SPLINE
SPL {X  -165.650, Y  +484.445, Z    +0.000, E1   +32.277, E3 +467467.662}
SPL {X  -165.650, Y  +481.524, Z    +0.000, E1   +31.089, E3 +467485.112}
SPL {X  -165.650, Y  +478.014, Z    +0.000, E1   +30.826, E3 +467498.720}
SPL {X  -165.650, Y  +474.473, Z    +0.000, E1   +30.943, E3 +467510.044}
SPL {X  -165.650, Y  +471.826, Z    +0.000, E1   +30.770, E3 +467520.228}
SPL {X  -165.650, Y  +467.753, Z    +0.000, E1   +30.878, E3 +467533.601}
SPL {X  -165.650, Y  +463.837, Z    +0.000, E1   +30.924, E3 +467546.535}
SPL {X  -165.650, Y  +461.106, Z    +0.000, E1   +30.916, E3 +467555.922}
SPL {X  -165.650, Y  +457.156, Z    +0.000, E1   +30.860, E3 +467569.999}
SPL {X  -165.650, Y  +453.156, Z    +0.000, E1   +30.934, E3 +467582.973}
SPL {X  -165.650, Y  +450.433, Z    +0.000, E1   +30.789, E3 +467593.328}
SPL {X  -165.650, Y  +447.097, Z    +0.000, E1   +30.843, E3 +467604.377}
SPL {X  -165.650, Y  +443.673, Z    +0.000, E1   +30.907, E3 +467615.684}
SPL {X  -165.650, Y  +439.486, Z    +0.000, E1   +30.857, E3 +467630.493}
SPL {X  -165.650, Y  +434.043, Z    +0.000, E1   +30.950, E3 +467648.510}
SPL {X  -165.650, Y  +430.419, Z    +0.000, E1   +30.895, E3 +467661.013}
SPL {X  -165.650, Y  +427.340, Z    +0.000, E1   +30.870, E3 +467671.839}
SPL {X  -165.650, Y  +422.641, Z    +0.000, E1   +30.884, E3 +467687.928}
SPL {X  -165.650, Y  +417.366, Z    +0.000, E1   +30.879, E3 +467706.034}
SPL {X  -165.650, Y  +412.139, Z    +0.000, E1   +30.870, E3 +467723.984}
SPL {X  -165.650, Y  +406.834, Z    +0.000, E1   +30.919, E3 +467741.812}
SPL {X  -165.650, Y  +402.516, Z    +0.000, E1   +30.874, E3 +467756.734}
SPL {X  -165.650, Y  +398.147, Z    +0.000, E1   +30.902, E3 +467771.613}
SPL {X  -165.650, Y  +394.694, Z    +0.000, E1   +30.805, E3 +467783.921}
SPL {X  -165.650, Y  +391.522, Z    +0.000, E1   +30.837, E3 +467794.602}
SPL {X  -165.650, Y  +387.533, Z    +0.000, E1   +30.858, E3 +467808.228}
SPL {X  -165.650, Y  +383.627, Z    +0.000, E1   +30.885, E3 +467821.289}
SPL {X  -165.650, Y  +380.752, Z    +0.000, E1   +30.927, E3 +467830.802}
SPL {X  -165.648, Y  +377.739, Z    +0.000, E1   +30.835, E3 +467841.812}
SPL {X  -165.594, Y  +374.183, Z    +0.000, E1   +30.878, E3 +467853.649}
SPL {X  -165.492, Y  +371.263, Z    +0.000, E1   +30.913, E3 +467863.344}
SPL {X  -165.379, Y  +369.027, Z    +0.000, E1   +30.727, E3 +467872.282}
SPL {X  -165.167, Y  +365.866, Z    +0.000, E1   +30.741, E3 +467883.056}
SPL {X  -164.892, Y  +362.671, Z    +0.000, E1   +30.830, E3 +467893.380}
SPL {X  -164.570, Y  +359.612, Z    +0.000, E1   +30.773, E3 +467904.193}
SPL {X  -164.104, Y  +355.923, Z    +0.000, E1   +30.626, E3 +467917.910}
SPL {X  -163.573, Y  +352.353, Z    +0.000, E1   +30.451, E3 +467931.174}
SPL {X  -162.476, Y  +346.230, Z    +0.000, E1   +31.677, E3 +467943.755}
SPL {X  -152.976, Y  +314.952, Z    +0.000, E1   +38.607, E3 +467992.720}
SPL {X  -137.967, Y  +286.821, Z    +0.000, E1   +43.969, E3 +468035.941}
ENDSPLINE

SPLINE
SPL {X  -153.316, Y  +315.777, Z    +0.000, E1   +33.140, E3 +468078.569}
SPL {X  -164.446, Y  +358.564, Z    +0.000, E1   +15.149, E3 +468043.780}
SPL {X  -165.379, Y  +369.025, Z    +0.000, E1    +9.158, E3 +468049.504}
SPL {X  -165.612, Y  +374.969, Z    +0.000, E1    +5.630, E3 +468052.180}
SPL {X  -165.650, Y  +383.362, Z    +0.000, E1    +0.177, E3 +468036.798}
SPL {X  -165.650, Y  +383.923, Z    +0.000, E1    -0.215, E3 +468049.956}
SPL {X  -165.650, Y  +388.083, Z    +0.000, E1    -3.355, E3 +468048.819}
SPL {X  -165.650, Y  +393.983, Z    +0.000, E1    -8.501, E3 +468045.218}
SPL {X  -165.650, Y  +402.241, Z    +0.000, E1   -16.711, E3 +468039.729}
SPL {X  -165.650, Y  +416.345, Z    +0.000, E1   -29.511, E3 +468039.521}
SPL {X  -165.650, Y  +422.331, Z    +0.000, E1   -27.760, E3 +468065.020}
SPL {X  -165.650, Y  +441.276, Z    +0.000, E1   -37.343, E3 +468074.877}
SPL {X  -165.650, Y  +462.890, Z    +0.000, E1   -40.484, E3 +468108.960}
ENDSPLINE

SPLINE
SPL {X  -165.650, Y  +446.920, Z    +0.000, E1   -31.238, E3 +468121.286}
ENDSPLINE

SPLINE
SPL {X  -165.650, Y  +447.935, Z    +0.000, E1   -30.213, E3 +468131.574}
SPL {X  -165.650, Y  +451.020, Z    +0.000, E1   -30.224, E3 +468142.394}
SPL {X  -165.650, Y  +454.519, Z    +0.000, E1   -30.374, E3 +468153.577}
SPL {X  -165.650, Y  +457.429, Z    +0.000, E1   -30.029, E3 +468166.278}
SPL {X  -165.650, Y  +461.678, Z    +0.000, E1   -30.426, E3 +468178.403}
SPL {X  -165.650, Y  +463.853, Z    +0.000, E1   -30.103, E3 +468188.243}
SPL {X  -165.650, Y  +468.397, Z    +0.000, E1   -30.302, E3 +468203.047}
SPL {X  -165.650, Y  +472.566, Z    +0.000, E1   -30.124, E3 +468218.756}
SPL {X  -165.650, Y  +476.540, Z    +0.000, E1   -30.193, E3 +468232.300}
SPL {X  -165.650, Y  +481.042, Z    +0.000, E1   -30.192, E3 +468248.245}
SPL {X  -165.650, Y  +485.236, Z    +0.000, E1   -30.294, E3 +468262.101}
SPL {X  -165.650, Y  +489.057, Z    +0.000, E1   -30.341, E3 +468275.307}
SPL {X  -165.650, Y  +491.647, Z    +0.000, E1   -29.894, E3 +468287.240}
SPL {X  -165.650, Y  +495.051, Z    +0.000, E1   -30.213, E3 +468297.169}
SPL {X  -165.650, Y  +498.418, Z    +0.000, E1   -30.282, E3 +468308.462}
SPL {X  -165.650, Y  +502.421, Z    +0.000, E1   -30.263, E3 +468322.819}
SPL {X  -165.650, Y  +506.344, Z    +0.000, E1   -30.129, E3 +468337.349}
SPL {X  -165.650, Y  +509.866, Z    +0.000, E1   -30.236, E3 +468349.018}
SPL {X  -165.650, Y  +513.685, Z    +0.000, E1   -30.234, E3 +468362.515}
SPL {X  -165.650, Y  +517.919, Z    +0.000, E1   -30.227, E3 +468377.421}
SPL {X  -165.650, Y  +521.521, Z    +0.000, E1   -30.210, E3 +468390.096}
SPL {X  -165.650, Y  +525.344, Z    +0.000, E1   -30.269, E3 +468403.202}
SPL {X  -165.650, Y  +528.152, Z    +0.000, E1   -29.991, E3 +468414.843}
SPL {X  -165.650, Y  +531.783, Z    +0.000, E1   -30.416, E3 +468424.736}
SPL {X  -165.650, Y  +534.115, Z    +0.000, E1   -30.089, E3 +468435.118}
SPL {X  -165.650, Y  +537.522, Z    +0.000, E1   -30.251, E3 +468446.033}
SPL {X  -165.650, Y  +540.621, Z    +0.000, E1   -30.014, E3 +468458.593}
SPL {X  -165.650, Y  +544.944, Z    +0.000, E1   -30.447, E3 +468470.793}
SPL {X  -165.650, Y  +548.549, Z    +0.000, E1   -30.216, E3 +468485.117}
SPL {X  -165.650, Y  +553.092, Z    +0.000, E1   -30.157, E3 +468501.459}
SPL {X  -165.650, Y  +556.274, Z    +0.000, E1   -30.127, E3 +468512.714}
SPL {X  -165.650, Y  +560.243, Z    +0.000, E1   -30.214, E3 +468526.380}
SPL {X  -165.650, Y  +565.528, Z    +0.000, E1   -30.192, E3 +468545.072}
SPL {X  -165.650, Y  +570.048, Z    +0.000, E1   -30.238, E3 +468560.503}
SPL {X  -165.650, Y  +573.110, Z    +0.000, E1   -30.057, E3 +468572.488}
SPL {X  -165.650, Y  +577.587, Z    +0.000, E1   -30.270, E3 +468586.927}
SPL {X  -165.650, Y  +581.190, Z    +0.000, E1   -30.107, E3 +468600.566}
SPL {X  -165.650, Y  +585.053, Z    +0.000, E1   -30.090, E3 +468614.436}
ENDSPLINE

SPLINE
SPL {X  -165.650, Y  +484.445, Z    +0.000, E1   +32.277, E3 +468631.841}
SPL {X  -165.650, Y  +481.524, Z    +0.000, E1   +31.089, E3 +468649.291}
SPL {X  -165.650, Y  +478.014, Z    +0.000, E1   +30.826, E3 +468662.899}
SPL {X  -165.650, Y  +474.473, Z    +0.000, E1   +30.943, E3 +468674.223}
SPL {X  -165.650, Y  +471.826, Z    +0.000, E1   +30.770, E3 +468684.407}
SPL {X  -165.650, Y  +467.753, Z    +0.000, E1   +30.878, E3 +468697.780}
SPL {X  -165.650, Y  +463.837, Z    +0.000, E1   +30.924, E3 +468710.714}
SPL {X  -165.650, Y  +461.106, Z    +0.000, E1   +30.916, E3 +468720.101}
SPL {X  -165.650, Y  +458.435, Z    +0.000, E1   +30.759, E3 +468730.309}
SPL {X  -165.650, Y  +454.220, Z    +0.000, E1   +30.954, E3 +468743.542}
SPL {X  -165.650, Y  +450.433, Z    +0.000, E1   +30.789, E3 +468757.507}
SPL {X  -165.650, Y  +447.097, Z    +0.000, E1   +30.843, E3 +468768.556}
SPL {X  -165.650, Y  +443.673, Z    +0.000, E1   +30.907, E3 +468779.863}
SPL {X  -165.650, Y  +440.976, Z    +0.000, E1   +30.719, E3 +468790.320}
SPL {X  -165.650, Y  +436.324, Z    +0.000, E1   +30.994, E3 +468804.606}
SPL {X  -165.650, Y  +432.765, Z    +0.000, E1   +30.831, E3 +468817.606}
SPL {X  -165.650, Y  +429.309, Z    +0.000, E1   +30.920, E3 +468828.947}
SPL {X  -165.650, Y  +424.918, Z    +0.000, E1   +30.862, E3 +468844.404}
SPL {X  -165.650, Y  +421.437, Z    +0.000, E1   +30.833, E3 +468856.373}
SPL {X  -165.650, Y  +417.366, Z    +0.000, E1   +30.879, E3 +468870.213}
SPL {X  -165.650, Y  +413.181, Z    +0.000, E1   +30.815, E3 +468884.811}
SPL {X  -165.650, Y  +408.547, Z    +0.000, E1   +30.964, E3 +468899.814}
SPL {X  -165.650, Y  +403.421, Z    +0.000, E1   +30.863, E3 +468918.031}
SPL {X  -165.650, Y  +398.147, Z    +0.000, E1   +30.902, E3 +468935.792}
SPL {X  -165.650, Y  +394.694, Z    +0.000, E1   +30.805, E3 +468948.100}
SPL {X  -165.650, Y  +391.522, Z    +0.000, E1   +30.837, E3 +468958.781}
SPL {X  -165.650, Y  +387.533, Z    +0.000, E1   +30.858, E3 +468972.407}
SPL {X  -165.650, Y  +383.627, Z    +0.000, E1   +30.885, E3 +468985.468}
SPL {X  -165.650, Y  +379.886, Z    +0.000, E1   +30.887, E3 +468998.356}
SPL {X  -165.614, Y  +375.058, Z    +0.000, E1   +30.905, E3 +469014.809}
SPL {X  -165.492, Y  +371.263, Z    +0.000, E1   +30.913, E3 +469027.523}
SPL {X  -165.379, Y  +369.027, Z    +0.000, E1   +30.727, E3 +469036.461}
SPL {X  -165.167, Y  +365.866, Z    +0.000, E1   +30.741, E3 +469047.235}
SPL {X  -164.892, Y  +362.671, Z    +0.000, E1   +30.830, E3 +469057.559}
SPL {X  -164.570, Y  +359.612, Z    +0.000, E1   +30.773, E3 +469068.372}
SPL {X  -164.104, Y  +355.923, Z    +0.000, E1   +30.626, E3 +469082.089}
SPL {X  -163.573, Y  +352.353, Z    +0.000, E1   +30.451, E3 +469095.353}
SPL {X  -162.476, Y  +346.230, Z    +0.000, E1   +31.677, E3 +469107.934}
SPL {X  -152.976, Y  +314.952, Z    +0.000, E1   +38.607, E3 +469156.899}
SPL {X  -137.967, Y  +286.821, Z    +0.000, E1   +43.969, E3 +469200.120}
ENDSPLINE

SPLINE
SPL {X  -153.316, Y  +315.777, Z    +0.000, E1   +33.140, E3 +469242.748}
SPL {X  -164.446, Y  +358.564, Z    +0.000, E1   +15.149, E3 +469207.959}
SPL {X  -165.510, Y  +371.680, Z    +0.000, E1    +7.684, E3 +469212.014}
SPL {X  -165.628, Y  +375.818, Z    +0.000, E1    +5.016, E3 +469219.944}
SPL {X  -165.650, Y  +383.362, Z    +0.000, E1    +0.177, E3 +469200.977}
SPL {X  -165.650, Y  +383.923, Z    +0.000, E1    -0.215, E3 +469214.135}
SPL {X  -165.650, Y  +388.083, Z    +0.000, E1    -3.355, E3 +469212.998}
SPL {X  -165.650, Y  +393.983, Z    +0.000, E1    -8.501, E3 +469209.397}
SPL {X  -165.650, Y  +402.241, Z    +0.000, E1   -16.711, E3 +469203.908}
SPL {X  -165.650, Y  +414.811, Z    +0.000, E1   -28.314, E3 +469203.439}
SPL {X  -165.650, Y  +423.479, Z    +0.000, E1   -29.012, E3 +469227.368}
SPL {X  -165.650, Y  +441.276, Z    +0.000, E1   -37.343, E3 +469239.056}
SPL {X  -165.650, Y  +462.890, Z    +0.000, E1   -40.484, E3 +469273.139}
ENDSPLINE

SPLINE
SPL {X  -165.650, Y  +446.920, Z    +0.000, E1   -31.238, E3 +469285.465}
ENDSPLINE

SPLINE
SPL {X  -165.650, Y  +447.935, Z    +0.000, E1   -30.213, E3 +469295.753}
SPL {X  -165.650, Y  +451.020, Z    +0.000, E1   -30.224, E3 +469306.573}
SPL {X  -165.650, Y  +454.519, Z    +0.000, E1   -30.374, E3 +469317.756}
SPL {X  -165.650, Y  +456.542, Z    +0.000, E1   -29.986, E3 +469327.500}
SPL {X  -165.650, Y  +460.618, Z    +0.000, E1   -30.298, E3 +469339.821}
SPL {X  -165.650, Y  +463.853, Z    +0.000, E1   -30.103, E3 +469352.422}
SPL {X  -165.650, Y  +468.397, Z    +0.000, E1   -30.302, E3 +469367.226}
SPL {X  -165.650, Y  +472.566, Z    +0.000, E1   -30.124, E3 +469382.935}
SPL {X  -165.650, Y  +475.265, Z    +0.000, E1   -30.034, E3 +469392.972}
SPL {X  -165.650, Y  +477.862, Z    +0.000, E1   -30.319, E3 +469400.164}
SPL {X  -165.650, Y  +481.042, Z    +0.000, E1   -30.192, E3 +469412.424}
SPL {X  -165.650, Y  +485.236, Z    +0.000, E1   -30.294, E3 +469426.280}
SPL {X  -165.650, Y  +488.041, Z    +0.000, E1   -30.253, E3 +469436.401}
SPL {X  -165.650, Y  +491.281, Z    +0.000, E1   -30.148, E3 +469448.539}
SPL {X  -165.650, Y  +495.051, Z    +0.000, E1   -30.213, E3 +469461.348}
SPL {X  -165.650, Y  +499.546, Z    +0.000, E1   -30.283, E3 +469476.791}
SPL {X  -165.650, Y  +503.544, Z    +0.000, E1   -30.247, E3 +469490.859}
SPL {X  -165.650, Y  +506.344, Z    +0.000, E1   -30.129, E3 +469501.528}
SPL {X  -165.650, Y  +510.660, Z    +0.000, E1   -30.223, E3 +469516.231}
SPL {X  -165.650, Y  +514.670, Z    +0.000, E1   -30.278, E3 +469529.741}
SPL {X  -165.650, Y  +517.919, Z    +0.000, E1   -30.227, E3 +469541.601}
SPL {X  -165.650, Y  +521.521, Z    +0.000, E1   -30.210, E3 +469554.275}
SPL {X  -165.650, Y  +525.344, Z    +0.000, E1   -30.269, E3 +469567.382}
SPL {X  -165.650, Y  +528.152, Z    +0.000, E1   -29.991, E3 +469579.022}
SPL {X  -165.650, Y  +531.783, Z    +0.000, E1   -30.416, E3 +469588.915}
SPL {X  -165.650, Y  +534.115, Z    +0.000, E1   -30.089, E3 +469599.297}
SPL {X  -165.650, Y  +537.522, Z    +0.000, E1   -30.251, E3 +469610.212}
SPL {X  -165.650, Y  +540.621, Z    +0.000, E1   -30.014, E3 +469622.773}
SPL {X  -165.650, Y  +544.944, Z    +0.000, E1   -30.447, E3 +469634.972}
SPL {X  -165.650, Y  +547.199, Z    +0.000, E1   -30.132, E3 +469644.946}
SPL {X  -165.650, Y  +550.512, Z    +0.000, E1   -30.197, E3 +469656.272}
SPL {X  -165.650, Y  +553.852, Z    +0.000, E1   -30.156, E3 +469668.212}
SPL {X  -165.650, Y  +557.277, Z    +0.000, E1   -30.150, E3 +469680.387}
SPL {X  -165.650, Y  +561.168, Z    +0.000, E1   -30.194, E3 +469693.768}
SPL {X  -165.650, Y  +564.449, Z    +0.000, E1   -30.167, E3 +469705.452}
SPL {X  -165.650, Y  +566.935, Z    +0.000, E1   -30.135, E3 +469714.357}
SPL {X  -165.650, Y  +570.048, Z    +0.000, E1   -30.238, E3 +469724.682}
SPL {X  -165.650, Y  +573.110, Z    +0.000, E1   -30.057, E3 +469736.667}
SPL {X  -165.650, Y  +577.587, Z    +0.000, E1   -30.270, E3 +469751.106}
SPL {X  -165.650, Y  +581.190, Z    +0.000, E1   -30.107, E3 +469764.745}
SPL {X  -165.650, Y  +585.053, Z    +0.000, E1   -30.090, E3 +469778.616}
ENDSPLINE

SPLINE
SPL {X  -165.650, Y  +484.445, Z    +0.000, E1   +32.277, E3 +469796.020}
SPL {X  -165.650, Y  +481.524, Z    +0.000, E1   +31.089, E3 +469813.471}
SPL {X  -165.650, Y  +478.014, Z    +0.000, E1   +30.826, E3 +469827.078}
SPL {X  -165.650, Y  +474.473, Z    +0.000, E1   +30.943, E3 +469838.403}
SPL {X  -165.650, Y  +471.826, Z    +0.000, E1   +30.770, E3 +469848.586}
SPL {X  -165.650, Y  +467.753, Z    +0.000, E1   +30.878, E3 +469861.960}
SPL {X  -165.650, Y  +463.837, Z    +0.000, E1   +30.924, E3 +469874.893}
SPL {X  -165.650, Y  +461.106, Z    +0.000, E1   +30.916, E3 +469884.280}
SPL {X  -165.650, Y  +458.435, Z    +0.000, E1   +30.759, E3 +469894.488}
SPL {X  -165.650, Y  +454.220, Z    +0.000, E1   +30.954, E3 +469907.721}
SPL {X  -165.650, Y  +450.433, Z    +0.000, E1   +30.789, E3 +469921.686}
SPL {X  -165.650, Y  +447.097, Z    +0.000, E1   +30.843, E3 +469932.735}
SPL {X  -165.650, Y  +443.673, Z    +0.000, E1   +30.907, E3 +469944.042}
SPL {X  -165.650, Y  +440.976, Z    +0.000, E1   +30.719, E3 +469954.499}
SPL {X  -165.650, Y  +437.973, Z    +0.000, E1   +30.928, E3 +469963.371}
SPL {X  -165.650, Y  +434.043, Z    +0.000, E1   +30.950, E3 +469976.868}
SPL {X  -165.650, Y  +430.419, Z    +0.000, E1   +30.895, E3 +469989.371}
SPL {X  -165.650, Y  +427.340, Z    +0.000, E1   +30.870, E3 +470000.197}
SPL {X  -165.650, Y  +422.641, Z    +0.000, E1   +30.884, E3 +470016.286}
SPL {X  -165.650, Y  +418.489, Z    +0.000, E1   +30.835, E3 +470030.669}
SPL {X  -165.650, Y  +414.127, Z    +0.000, E1   +30.869, E3 +470045.577}
SPL {X  -165.650, Y  +408.547, Z    +0.000, E1   +30.964, E3 +470063.993}
SPL {X  -165.650, Y  +405.433, Z    +0.000, E1   +30.730, E3 +470075.970}
SPL {X  -165.650, Y  +402.516, Z    +0.000, E1   +30.874, E3 +470085.093}
SPL {X  -165.650, Y  +398.147, Z    +0.000, E1   +30.902, E3 +470099.971}
SPL {X  -165.650, Y  +394.694, Z    +0.000, E1   +30.805, E3 +470112.279}
SPL {X  -165.650, Y  +391.522, Z    +0.000, E1   +30.837, E3 +470122.960}
SPL {X  -165.650, Y  +387.533, Z    +0.000, E1   +30.858, E3 +470136.586}
SPL {X  -165.650, Y  +383.627, Z    +0.000, E1   +30.885, E3 +470149.647}
SPL {X  -165.650, Y  +379.886, Z    +0.000, E1   +30.887, E3 +470162.535}
SPL {X  -165.614, Y  +375.058, Z    +0.000, E1   +30.905, E3 +470178.988}
SPL {X  -165.492, Y  +371.263, Z    +0.000, E1   +30.913, E3 +470191.702}
SPL {X  -165.379, Y  +369.027, Z    +0.000, E1   +30.727, E3 +470200.640}
SPL {X  -165.167, Y  +365.866, Z    +0.000, E1   +30.741, E3 +470211.415}
SPL {X  -164.892, Y  +362.671, Z    +0.000, E1   +30.830, E3 +470221.739}
SPL {X  -164.570, Y  +359.612, Z    +0.000, E1   +30.773, E3 +470232.551}
SPL {X  -164.104, Y  +355.923, Z    +0.000, E1   +30.626, E3 +470246.268}
SPL {X  -163.573, Y  +352.353, Z    +0.000, E1   +30.451, E3 +470259.532}
SPL {X  -162.976, Y  +348.856, Z    +0.000, E1   +30.757, E3 +470269.456}
SPL {X  -161.497, Y  +341.640, Z    +0.000, E1   +33.276, E3 +470276.734}
SPL {X  -152.976, Y  +314.952, Z    +0.000, E1   +38.607, E3 +470321.078}
SPL {X  -137.967, Y  +286.821, Z    +0.000, E1   +43.969, E3 +470364.300}
ENDSPLINE

SPLINE
SPL {X  -149.143, Y  +306.414, Z    +0.000, E1   +36.361, E3 +470415.432}
SPL {X  -164.268, Y  +357.145, Z    +0.000, E1   +15.880, E3 +470373.191}
SPL {X  -165.379, Y  +369.025, Z    +0.000, E1    +9.158, E3 +470377.863}
SPL {X  -165.612, Y  +374.969, Z    +0.000, E1    +5.630, E3 +470380.538}
SPL {X  -165.650, Y  +383.362, Z    +0.000, E1    +0.177, E3 +470365.157}
SPL {X  -165.650, Y  +383.923, Z    +0.000, E1    -0.215, E3 +470378.314}
SPL {X  -165.650, Y  +388.083, Z    +0.000, E1    -3.355, E3 +470377.177}
SPL {X  -165.650, Y  +393.983, Z    +0.000, E1    -8.501, E3 +470373.576}
SPL {X  -165.650, Y  +402.241, Z    +0.000, E1   -16.711, E3 +470368.087}
SPL {X  -165.650, Y  +416.345, Z    +0.000, E1   -29.511, E3 +470367.879}
SPL {X  -165.650, Y  +422.331, Z    +0.000, E1   -27.760, E3 +470393.378}
SPL {X  -165.650, Y  +441.276, Z    +0.000, E1   -37.343, E3 +470403.236}
SPL {X  -165.650, Y  +462.890, Z    +0.000, E1   -40.484, E3 +470437.318}
ENDSPLINE

SPLINE
SPL {X  -165.650, Y  +446.920, Z    +0.000, E1   -31.238, E3 +470449.644}
ENDSPLINE

SPLINE
SPL {X  -165.650, Y  +447.935, Z    +0.000, E1   -30.213, E3 +470459.932}
SPL {X  -165.650, Y  +451.020, Z    +0.000, E1   -30.224, E3 +470470.753}
SPL {X  -165.650, Y  +454.519, Z    +0.000, E1   -30.374, E3 +470481.935}
SPL {X  -165.650, Y  +456.542, Z    +0.000, E1   -29.986, E3 +470491.680}
SPL {X  -165.650, Y  +460.618, Z    +0.000, E1   -30.298, E3 +470504.000}
SPL {X  -165.650, Y  +463.853, Z    +0.000, E1   -30.103, E3 +470516.601}
SPL {X  -165.650, Y  +468.397, Z    +0.000, E1   -30.302, E3 +470531.405}
SPL {X  -165.650, Y  +472.566, Z    +0.000, E1   -30.124, E3 +470547.114}
SPL {X  -165.650, Y  +476.540, Z    +0.000, E1   -30.193, E3 +470560.658}
SPL {X  -165.650, Y  +480.320, Z    +0.000, E1   -30.163, E3 +470574.136}
SPL {X  -165.650, Y  +484.477, Z    +0.000, E1   -30.274, E3 +470588.025}
SPL {X  -165.650, Y  +488.041, Z    +0.000, E1   -30.253, E3 +470600.580}
SPL {X  -165.650, Y  +491.281, Z    +0.000, E1   -30.148, E3 +470612.719}
SPL {X  -165.650, Y  +495.051, Z    +0.000, E1   -30.213, E3 +470625.527}
SPL {X  -165.650, Y  +499.546, Z    +0.000, E1   -30.283, E3 +470640.970}
SPL {X  -165.650, Y  +503.544, Z    +0.000, E1   -30.247, E3 +470655.038}
SPL {X  -165.650, Y  +506.344, Z    +0.000, E1   -30.129, E3 +470665.707}
SPL {X  -165.650, Y  +509.866, Z    +0.000, E1   -30.236, E3 +470677.376}
SPL {X  -165.650, Y  +513.685, Z    +0.000, E1   -30.234, E3 +470690.873}
SPL {X  -165.650, Y  +517.919, Z    +0.000, E1   -30.227, E3 +470705.780}
SPL {X  -165.650, Y  +521.521, Z    +0.000, E1   -30.210, E3 +470718.454}
SPL {X  -165.650, Y  +525.344, Z    +0.000, E1   -30.269, E3 +470731.561}
SPL {X  -165.650, Y  +528.152, Z    +0.000, E1   -29.991, E3 +470743.202}
SPL {X  -165.650, Y  +531.783, Z    +0.000, E1   -30.416, E3 +470753.094}
SPL {X  -165.650, Y  +534.115, Z    +0.000, E1   -30.089, E3 +470763.476}
SPL {X  -165.650, Y  +537.522, Z    +0.000, E1   -30.251, E3 +470774.391}
SPL {X  -165.650, Y  +540.621, Z    +0.000, E1   -30.014, E3 +470786.952}
SPL {X  -165.650, Y  +544.944, Z    +0.000, E1   -30.447, E3 +470799.151}
SPL {X  -165.650, Y  +547.199, Z    +0.000, E1   -30.132, E3 +470809.125}
SPL {X  -165.650, Y  +550.512, Z    +0.000, E1   -30.197, E3 +470820.451}
SPL {X  -165.650, Y  +553.852, Z    +0.000, E1   -30.156, E3 +470832.391}
SPL {X  -165.650, Y  +557.277, Z    +0.000, E1   -30.150, E3 +470844.566}
SPL {X  -165.650, Y  +561.168, Z    +0.000, E1   -30.194, E3 +470857.947}
SPL {X  -165.650, Y  +565.528, Z    +0.000, E1   -30.192, E3 +470873.430}
SPL {X  -165.650, Y  +570.048, Z    +0.000, E1   -30.238, E3 +470888.861}
SPL {X  -165.650, Y  +573.110, Z    +0.000, E1   -30.057, E3 +470900.846}
SPL {X  -165.650, Y  +577.587, Z    +0.000, E1   -30.270, E3 +470915.285}
SPL {X  -165.650, Y  +581.190, Z    +0.000, E1   -30.107, E3 +470928.925}
SPL {X  -165.650, Y  +585.053, Z    +0.000, E1   -30.090, E3 +470942.795}
ENDSPLINE

SPLINE
SPL {X  -165.650, Y  +484.445, Z    +0.000, E1   +32.277, E3 +470960.199}
SPL {X  -165.650, Y  +481.524, Z    +0.000, E1   +31.089, E3 +470977.650}
SPL {X  -165.650, Y  +478.014, Z    +0.000, E1   +30.826, E3 +470991.257}
SPL {X  -165.650, Y  +474.473, Z    +0.000, E1   +30.943, E3 +471002.582}
SPL {X  -165.650, Y  +471.826, Z    +0.000, E1   +30.770, E3 +471012.765}
SPL {X  -165.650, Y  +467.753, Z    +0.000, E1   +30.878, E3 +471026.139}
SPL {X  -165.650, Y  +463.837, Z    +0.000, E1   +30.924, E3 +471039.073}
SPL {X  -165.650, Y  +461.106, Z    +0.000, E1   +30.916, E3 +471048.459}
SPL {X  -165.650, Y  +457.156, Z    +0.000, E1   +30.860, E3 +471062.536}
SPL {X  -165.650, Y  +453.156, Z    +0.000, E1   +30.934, E3 +471075.510}
SPL {X  -165.650, Y  +450.433, Z    +0.000, E1   +30.789, E3 +471085.865}
SPL {X  -165.650, Y  +447.097, Z    +0.000, E1   +30.843, E3 +471096.914}
SPL {X  -165.650, Y  +443.673, Z    +0.000, E1   +30.907, E3 +471108.221}
SPL {X  -165.650, Y  +439.486, Z    +0.000, E1   +30.857, E3 +471123.031}
SPL {X  -165.650, Y  +435.146, Z    +0.000, E1   +30.969, E3 +471136.950}
SPL {X  -165.650, Y  +432.765, Z    +0.000, E1   +30.831, E3 +471145.965}
SPL {X  -165.650, Y  +429.309, Z    +0.000, E1   +30.920, E3 +471157.305}
SPL {X  -165.650, Y  +424.918, Z    +0.000, E1   +30.862, E3 +471172.763}
SPL {X  -165.650, Y  +421.437, Z    +0.000, E1   +30.833, E3 +471184.731}
SPL {X  -165.650, Y  +417.366, Z    +0.000, E1   +30.879, E3 +471198.571}
SPL {X  -165.650, Y  +413.181, Z    +0.000, E1   +30.815, E3 +471213.169}
SPL {X  -165.650, Y  +408.547, Z    +0.000, E1   +30.964, E3 +471228.172}
SPL {X  -165.650, Y  +403.421, Z    +0.000, E1   +30.863, E3 +471246.390}
SPL {X  -165.650, Y  +399.681, Z    +0.000, E1   +30.933, E3 +471258.472}
SPL {X  -165.650, Y  +396.018, Z    +0.000, E1   +30.861, E3 +471271.782}
SPL {X  -165.650, Y  +391.522, Z    +0.000, E1   +30.837, E3 +471287.139}
SPL {X  -165.650, Y  +387.533, Z    +0.000, E1   +30.858, E3 +471300.766}
SPL {X  -165.650, Y  +383.627, Z    +0.000, E1   +30.885, E3 +471313.826}
SPL {X  -165.650, Y  +380.752, Z    +0.000, E1   +30.927, E3 +471323.340}
SPL {X  -165.648, Y  +377.739, Z    +0.000, E1   +30.835, E3 +471334.349}
SPL {X  -165.594, Y  +374.183, Z    +0.000, E1   +30.878, E3 +471346.186}
SPL {X  -165.429, Y  +369.945, Z    +0.000, E1   +30.850, E3 +471361.061}
SPL {X  -165.167, Y  +365.866, Z    +0.000, E1   +30.741, E3 +471375.594}
SPL {X  -164.892, Y  +362.671, Z    +0.000, E1   +30.830, E3 +471385.918}
SPL {X  -164.570, Y  +359.612, Z    +0.000, E1   +30.773, E3 +471396.730}
SPL {X  -164.287, Y  +357.291, Z    +0.000, E1   +30.513, E3 +471406.360}
SPL {X  -163.720, Y  +353.284, Z    +0.000, E1   +30.592, E3 +471419.807}
SPL {X  -162.976, Y  +348.856, Z    +0.000, E1   +30.757, E3 +471433.635}
SPL {X  -161.497, Y  +341.640, Z    +0.000, E1   +33.276, E3 +471440.913}
SPL {X  -152.976, Y  +314.952, Z    +0.000, E1   +38.607, E3 +471485.258}
SPL {X  -137.967, Y  +286.821, Z    +0.000, E1   +43.969, E3 +471528.479}
ENDSPLINE

SPLINE
SPL {X  -149.143, Y  +306.414, Z    +0.000, E1   +36.361, E3 +471579.611}
SPL {X  -164.268, Y  +357.145, Z    +0.000, E1   +15.880, E3 +471537.370}
SPL {X  -165.379, Y  +369.025, Z    +0.000, E1    +9.158, E3 +471542.042}
SPL {X  -165.612, Y  +374.969, Z    +0.000, E1    +5.630, E3 +471544.717}
SPL {X  -165.650, Y  +383.362, Z    +0.000, E1    +0.177, E3 +471529.336}
SPL {X  -165.650, Y  +383.923, Z    +0.000, E1    -0.215, E3 +471542.493}
SPL {X  -165.650, Y  +388.083, Z    +0.000, E1    -3.355, E3 +471541.357}
SPL {X  -165.650, Y  +393.983, Z    +0.000, E1    -8.501, E3 +471537.755}
SPL {X  -165.650, Y  +402.241, Z    +0.000, E1   -16.711, E3 +471532.267}
SPL {X  -165.650, Y  +416.345, Z    +0.000, E1   -29.511, E3 +471532.059}
SPL {X  -165.650, Y  +422.331, Z    +0.000, E1   -27.760, E3 +471557.558}
SPL {X  -165.650, Y  +441.276, Z    +0.000, E1   -37.343, E3 +471567.415}
SPL {X  -165.650, Y  +462.890, Z    +0.000, E1   -40.484, E3 +471601.498}
ENDSPLINE

SPLINE
SPL {X  -165.650, Y  +446.920, Z    +0.000, E1   -31.238, E3 +471613.823}
ENDSPLINE

SPLINE
SPL {X  -165.650, Y  +447.935, Z    +0.000, E1   -30.213, E3 +471624.111}
SPL {X  -165.650, Y  +451.020, Z    +0.000, E1   -30.224, E3 +471634.932}
SPL {X  -165.650, Y  +454.519, Z    +0.000, E1   -30.374, E3 +471646.114}
SPL {X  -165.650, Y  +457.429, Z    +0.000, E1   -30.029, E3 +471658.816}
SPL {X  -165.650, Y  +461.678, Z    +0.000, E1   -30.426, E3 +471670.940}
SPL {X  -165.650, Y  +463.853, Z    +0.000, E1   -30.103, E3 +471680.780}
SPL {X  -165.650, Y  +467.246, Z    +0.000, E1   -30.279, E3 +471691.510}
SPL {X  -165.650, Y  +469.780, Z    +0.000, E1   -30.237, E3 +471700.636}
SPL {X  -165.650, Y  +472.566, Z    +0.000, E1   -30.124, E3 +471711.293}
SPL {X  -165.650, Y  +475.265, Z    +0.000, E1   -30.034, E3 +471721.331}
SPL {X  -165.650, Y  +477.862, Z    +0.000, E1   -30.319, E3 +471728.522}
SPL {X  -165.650, Y  +481.042, Z    +0.000, E1   -30.192, E3 +471740.783}
SPL {X  -165.650, Y  +485.236, Z    +0.000, E1   -30.294, E3 +471754.638}
SPL {X  -165.650, Y  +488.041, Z    +0.000, E1   -30.253, E3 +471764.759}
SPL {X  -165.650, Y  +491.281, Z    +0.000, E1   -30.148, E3 +471776.898}
SPL {X  -165.650, Y  +495.051, Z    +0.000, E1   -30.213, E3 +471789.706}
SPL {X  -165.650, Y  +499.546, Z    +0.000, E1   -30.283, E3 +471805.149}
SPL {X  -165.650, Y  +503.544, Z    +0.000, E1   -30.247, E3 +471819.217}
SPL {X  -165.650, Y  +506.344, Z    +0.000, E1   -30.129, E3 +471829.886}
SPL {X  -165.650, Y  +509.866, Z    +0.000, E1   -30.236, E3 +471841.555}
SPL {X  -165.650, Y  +513.685, Z    +0.000, E1   -30.234, E3 +471855.052}
SPL {X  -165.650, Y  +517.919, Z    +0.000, E1   -30.227, E3 +471869.959}
SPL {X  -165.650, Y  +521.521, Z    +0.000, E1   -30.210, E3 +471882.634}
SPL {X  -165.650, Y  +525.344, Z    +0.000, E1   -30.269, E3 +471895.740}
SPL {X  -165.650, Y  +528.152, Z    +0.000, E1   -29.991, E3 +471907.381}
SPL {X  -165.650, Y  +531.783, Z    +0.000, E1   -30.416, E3 +471917.273}
SPL {X  -165.650, Y  +534.115, Z    +0.000, E1   -30.089, E3 +471927.656}
SPL {X  -165.650, Y  +537.522, Z    +0.000, E1   -30.251, E3 +471938.570}
SPL {X  -165.650, Y  +540.621, Z    +0.000, E1   -30.014, E3 +471951.131}
SPL {X  -165.650, Y  +544.944, Z    +0.000, E1   -30.447, E3 +471963.330}
SPL {X  -165.650, Y  +547.199, Z    +0.000, E1   -30.132, E3 +471973.304}
SPL {X  -165.650, Y  +550.512, Z    +0.000, E1   -30.197, E3 +471984.630}
SPL {X  -165.650, Y  +553.852, Z    +0.000, E1   -30.156, E3 +471996.571}
SPL {X  -165.650, Y  +557.277, Z    +0.000, E1   -30.150, E3 +472008.745}
SPL {X  -165.650, Y  +561.168, Z    +0.000, E1   -30.194, E3 +472022.126}
SPL {X  -165.650, Y  +564.449, Z    +0.000, E1   -30.167, E3 +472033.810}
SPL {X  -165.650, Y  +566.935, Z    +0.000, E1   -30.135, E3 +472042.715}
SPL {X  -165.650, Y  +570.048, Z    +0.000, E1   -30.238, E3 +472053.040}
SPL {X  -165.650, Y  +573.110, Z    +0.000, E1   -30.057, E3 +472065.025}
SPL {X  -165.650, Y  +577.587, Z    +0.000, E1   -30.270, E3 +472079.464}
SPL {X  -165.650, Y  +581.190, Z    +0.000, E1   -30.107, E3 +472093.104}
SPL {X  -165.650, Y  +585.053, Z    +0.000, E1   -30.090, E3 +472106.974}
ENDSPLINE

SPLINE
SPL {X  -165.650, Y  +484.445, Z    +0.000, E1   +32.277, E3 +472124.378}
SPL {X  -165.650, Y  +481.524, Z    +0.000, E1   +31.089, E3 +472141.829}
SPL {X  -165.650, Y  +478.014, Z    +0.000, E1   +30.826, E3 +472155.436}
SPL {X  -165.650, Y  +474.473, Z    +0.000, E1   +30.943, E3 +472166.761}
SPL {X  -165.650, Y  +471.826, Z    +0.000, E1   +30.770, E3 +472176.944}
SPL {X  -165.650, Y  +467.753, Z    +0.000, E1   +30.878, E3 +472190.318}
SPL {X  -165.650, Y  +463.837, Z    +0.000, E1   +30.924, E3 +472203.252}
SPL {X  -165.650, Y  +461.106, Z    +0.000, E1   +30.916, E3 +472212.639}
SPL {X  -165.650, Y  +458.435, Z    +0.000, E1   +30.759, E3 +472222.847}
SPL {X  -165.650, Y  +454.220, Z    +0.000, E1   +30.954, E3 +472236.080}
SPL {X  -165.650, Y  +450.433, Z    +0.000, E1   +30.789, E3 +472250.044}
SPL {X  -165.650, Y  +447.097, Z    +0.000, E1   +30.843, E3 +472261.093}
SPL {X  -165.650, Y  +443.673, Z    +0.000, E1   +30.907, E3 +472272.401}
SPL {X  -165.650, Y  +440.976, Z    +0.000, E1   +30.719, E3 +472282.857}
SPL {X  -165.650, Y  +436.324, Z    +0.000, E1   +30.994, E3 +472297.144}
SPL {X  -165.650, Y  +432.765, Z    +0.000, E1   +30.831, E3 +472310.144}
SPL {X  -165.650, Y  +429.309, Z    +0.000, E1   +30.920, E3 +472321.484}
SPL {X  -165.650, Y  +424.918, Z    +0.000, E1   +30.862, E3 +472336.942}
SPL {X  -165.650, Y  +421.437, Z    +0.000, E1   +30.833, E3 +472348.910}
SPL {X  -165.650, Y  +418.489, Z    +0.000, E1   +30.835, E3 +472359.027}
SPL {X  -165.650, Y  +414.127, Z    +0.000, E1   +30.869, E3 +472373.935}
SPL {X  -165.650, Y  +408.547, Z    +0.000, E1   +30.964, E3 +472392.351}
SPL {X  -165.650, Y  +405.433, Z    +0.000, E1   +30.730, E3 +472404.328}
SPL {X  -165.650, Y  +402.516, Z    +0.000, E1   +30.874, E3 +472413.451}
SPL {X  -165.650, Y  +398.147, Z    +0.000, E1   +30.902, E3 +472428.329}
SPL {X  -165.650, Y  +394.694, Z    +0.000, E1   +30.805, E3 +472440.638}
SPL {X  -165.650, Y  +391.522, Z    +0.000, E1   +30.837, E3 +472451.318}
SPL {X  -165.650, Y  +387.533, Z    +0.000, E1   +30.858, E3 +472464.945}
SPL {X  -165.650, Y  +383.627, Z    +0.000, E1   +30.885, E3 +472478.005}
SPL {X  -165.650, Y  +379.886, Z    +0.000, E1   +30.887, E3 +472490.893}
SPL {X  -165.614, Y  +375.058, Z    +0.000, E1   +30.905, E3 +472507.346}
SPL {X  -165.492, Y  +371.263, Z    +0.000, E1   +30.913, E3 +472520.060}
SPL {X  -165.379, Y  +369.027, Z    +0.000, E1   +30.727, E3 +472528.999}
SPL {X  -165.167, Y  +365.866, Z    +0.000, E1   +30.741, E3 +472539.773}
SPL {X  -164.892, Y  +362.671, Z    +0.000, E1   +30.830, E3 +472550.097}
SPL {X  -164.570, Y  +359.612, Z    +0.000, E1   +30.773, E3 +472560.909}
SPL {X  -164.104, Y  +355.923, Z    +0.000, E1   +30.626, E3 +472574.626}
SPL {X  -163.573, Y  +352.353, Z    +0.000, E1   +30.451, E3 +472587.891}
SPL {X  -162.476, Y  +346.230, Z    +0.000, E1   +31.677, E3 +472600.472}
SPL {X  -152.976, Y  +314.952, Z    +0.000, E1   +38.607, E3 +472649.437}
SPL {X  -137.967, Y  +286.821, Z    +0.000, E1   +43.969, E3 +472692.658}
ENDSPLINE

SPLINE
SPL {X  -149.143, Y  +306.414, Z    +0.000, E1   +36.361, E3 +472743.790}
SPL {X  -164.268, Y  +357.145, Z    +0.000, E1   +15.880, E3 +472701.549}
SPL {X  -165.510, Y  +371.680, Z    +0.000, E1    +7.684, E3 +472704.552}
SPL {X  -165.628, Y  +375.818, Z    +0.000, E1    +5.016, E3 +472712.481}
SPL {X  -165.650, Y  +383.362, Z    +0.000, E1    +0.177, E3 +472693.515}
SPL {X  -165.650, Y  +383.923, Z    +0.000, E1    -0.215, E3 +472706.672}
SPL {X  -165.650, Y  +388.083, Z    +0.000, E1    -3.355, E3 +472705.536}
SPL {X  -165.650, Y  +393.983, Z    +0.000, E1    -8.501, E3 +472701.934}
SPL {X  -165.650, Y  +402.241, Z    +0.000, E1   -16.711, E3 +472696.446}
SPL {X  -165.650, Y  +416.345, Z    +0.000, E1   -29.511, E3 +472696.238}
SPL {X  -165.650, Y  +422.331, Z    +0.000, E1   -27.760, E3 +472721.737}
SPL {X  -165.650, Y  +441.276, Z    +0.000, E1   -37.343, E3 +472731.594}
SPL {X  -165.650, Y  +462.890, Z    +0.000, E1   -40.484, E3 +472765.677}
ENDSPLINE

SPLINE
SPL {X  -165.650, Y  +446.920, Z    +0.000, E1   -31.238, E3 +472778.002}
ENDSPLINE

SPLINE
SPL {X  -165.650, Y  +447.935, Z    +0.000, E1   -30.213, E3 +472788.290}
SPL {X  -165.650, Y  +451.020, Z    +0.000, E1   -30.224, E3 +472799.111}
SPL {X  -165.650, Y  +454.519, Z    +0.000, E1   -30.374, E3 +472810.293}
SPL {X  -165.650, Y  +456.542, Z    +0.000, E1   -29.986, E3 +472820.038}
SPL {X  -165.650, Y  +460.618, Z    +0.000, E1   -30.298, E3 +472832.358}
SPL {X  -165.650, Y  +463.853, Z    +0.000, E1   -30.103, E3 +472844.959}
SPL {X  -165.650, Y  +468.397, Z    +0.000, E1   -30.302, E3 +472859.763}
SPL {X  -165.650, Y  +472.566, Z    +0.000, E1   -30.124, E3 +472875.472}
SPL {X  -165.650, Y  +475.265, Z    +0.000, E1   -30.034, E3 +472885.510}
SPL {X  -165.650, Y  +477.862, Z    +0.000, E1   -30.319, E3 +472892.701}
SPL {X  -165.650, Y  +481.042, Z    +0.000, E1   -30.192, E3 +472904.962}
SPL {X  -165.650, Y  +485.236, Z    +0.000, E1   -30.294, E3 +472918.817}
SPL {X  -165.650, Y  +488.041, Z    +0.000, E1   -30.253, E3 +472928.939}
SPL {X  -165.650, Y  +491.281, Z    +0.000, E1   -30.148, E3 +472941.077}
SPL {X  -165.650, Y  +495.051, Z    +0.000, E1   -30.213, E3 +472953.885}
SPL {X  -165.650, Y  +499.546, Z    +0.000, E1   -30.283, E3 +472969.328}
SPL {X  -165.650, Y  +503.544, Z    +0.000, E1   -30.247, E3 +472983.397}
SPL {X  -165.650, Y  +506.344, Z    +0.000, E1   -30.129, E3 +472994.065}
SPL {X  -165.650, Y  +510.660, Z    +0.000, E1   -30.223, E3 +473008.769}
SPL {X  -165.650, Y  +514.670, Z    +0.000, E1   -30.278, E3 +473022.278}
SPL {X  -165.650, Y  +517.919, Z    +0.000, E1   -30.227, E3 +473034.138}
SPL {X  -165.650, Y  +521.521, Z    +0.000, E1   -30.210, E3 +473046.813}
SPL {X  -165.650, Y  +525.344, Z    +0.000, E1   -30.269, E3 +473059.919}
SPL {X  -165.650, Y  +528.152, Z    +0.000, E1   -29.991, E3 +473071.560}
SPL {X  -165.650, Y  +531.783, Z    +0.000, E1   -30.416, E3 +473081.453}
SPL {X  -165.650, Y  +534.115, Z    +0.000, E1   -30.089, E3 +473091.835}
SPL {X  -165.650, Y  +537.522, Z    +0.000, E1   -30.251, E3 +473102.749}
SPL {X  -165.650, Y  +540.621, Z    +0.000, E1   -30.014, E3 +473115.310}
SPL {X  -165.650, Y  +544.944, Z    +0.000, E1   -30.447, E3 +473127.510}
SPL {X  -165.650, Y  +547.199, Z    +0.000, E1   -30.132, E3 +473137.483}
SPL {X  -165.650, Y  +550.512, Z    +0.000, E1   -30.197, E3 +473148.809}
SPL {X  -165.650, Y  +553.852, Z    +0.000, E1   -30.156, E3 +473160.750}
SPL {X  -165.650, Y  +557.277, Z    +0.000, E1   -30.150, E3 +473172.924}
SPL {X  -165.650, Y  +561.168, Z    +0.000, E1   -30.194, E3 +473186.306}
SPL {X  -165.650, Y  +565.528, Z    +0.000, E1   -30.192, E3 +473201.788}
SPL {X  -165.650, Y  +570.048, Z    +0.000, E1   -30.238, E3 +473217.219}
SPL {X  -165.650, Y  +573.110, Z    +0.000, E1   -30.057, E3 +473229.204}
SPL {X  -165.650, Y  +577.587, Z    +0.000, E1   -30.270, E3 +473243.643}
SPL {X  -165.650, Y  +581.190, Z    +0.000, E1   -30.107, E3 +473257.283}
SPL {X  -165.650, Y  +585.053, Z    +0.000, E1   -30.090, E3 +473271.153}
ENDSPLINE

SPLINE
SPL {X  -165.650, Y  +484.445, Z    +0.000, E1   +32.277, E3 +473288.557}
SPL {X  -165.650, Y  +481.524, Z    +0.000, E1   +31.089, E3 +473306.008}
SPL {X  -165.650, Y  +478.014, Z    +0.000, E1   +30.826, E3 +473319.615}
SPL {X  -165.650, Y  +474.473, Z    +0.000, E1   +30.943, E3 +473330.940}
SPL {X  -165.650, Y  +470.376, Z    +0.000, E1   +30.888, E3 +473345.469}
SPL {X  -165.650, Y  +465.146, Z    +0.000, E1   +30.883, E3 +473363.400}
SPL {X  -165.650, Y  +461.106, Z    +0.000, E1   +30.916, E3 +473376.818}
SPL {X  -165.650, Y  +458.435, Z    +0.000, E1   +30.759, E3 +473387.026}
SPL {X  -165.650, Y  +454.220, Z    +0.000, E1   +30.954, E3 +473400.259}
SPL {X  -165.650, Y  +450.433, Z    +0.000, E1   +30.789, E3 +473414.224}
SPL {X  -165.650, Y  +447.097, Z    +0.000, E1   +30.843, E3 +473425.272}
SPL {X  -165.650, Y  +443.673, Z    +0.000, E1   +30.907, E3 +473436.580}
SPL {X  -165.650, Y  +440.976, Z    +0.000, E1   +30.719, E3 +473447.036}
SPL {X  -165.650, Y  +436.324, Z    +0.000, E1   +30.994, E3 +473461.323}
SPL {X  -165.650, Y  +432.765, Z    +0.000, E1   +30.831, E3 +473474.323}
SPL {X  -165.650, Y  +429.309, Z    +0.000, E1   +30.920, E3 +473485.664}
SPL {X  -165.650, Y  +424.918, Z    +0.000, E1   +30.862, E3 +473501.121}
SPL {X  -165.650, Y  +421.437, Z    +0.000, E1   +30.833, E3 +473513.089}
SPL {X  -165.650, Y  +417.366, Z    +0.000, E1   +30.879, E3 +473526.930}
SPL {X  -165.650, Y  +412.139, Z    +0.000, E1   +30.870, E3 +473544.879}
SPL {X  -165.650, Y  +406.834, Z    +0.000, E1   +30.919, E3 +473562.708}
SPL {X  -165.650, Y  +402.516, Z    +0.000, E1   +30.874, E3 +473577.630}
SPL {X  -165.650, Y  +398.147, Z    +0.000, E1   +30.902, E3 +473592.508}
SPL {X  -165.650, Y  +394.694, Z    +0.000, E1   +30.805, E3 +473604.817}
SPL {X  -165.650, Y  +391.522, Z    +0.000, E1   +30.837, E3 +473615.498}
SPL {X  -165.650, Y  +387.533, Z    +0.000, E1   +30.858, E3 +473629.124}
SPL {X  -165.650, Y  +383.627, Z    +0.000, E1   +30.885, E3 +473642.184}
SPL {X  -165.650, Y  +380.752, Z    +0.000, E1   +30.927, E3 +473651.698}
SPL {X  -165.648, Y  +377.739, Z    +0.000, E1   +30.835, E3 +473662.707}
SPL {X  -165.594, Y  +374.183, Z    +0.000, E1   +30.878, E3 +473674.544}
SPL {X  -165.492, Y  +371.263, Z    +0.000, E1   +30.913, E3 +473684.239}
SPL {X  -165.379, Y  +369.027, Z    +0.000, E1   +30.727, E3 +473693.178}
SPL {X  -165.167, Y  +365.866, Z    +0.000, E1   +30.741, E3 +473703.952}
SPL {X  -164.892, Y  +362.671, Z    +0.000, E1   +30.830, E3 +473714.276}
SPL {X  -164.570, Y  +359.612, Z    +0.000, E1   +30.773, E3 +473725.089}
SPL {X  -164.104, Y  +355.923, Z    +0.000, E1   +30.626, E3 +473738.805}
SPL {X  -163.573, Y  +352.353, Z    +0.000, E1   +30.451, E3 +473752.070}
SPL {X  -162.476, Y  +346.230, Z    +0.000, E1   +31.677, E3 +473764.651}
SPL {X  -152.976, Y  +314.952, Z    +0.000, E1   +38.607, E3 +473813.616}
SPL {X  -137.967, Y  +286.821, Z    +0.000, E1   +43.969, E3 +473856.837}
ENDSPLINE

SPLINE
SPL {X  -153.316, Y  +315.777, Z    +0.000, E1   +33.140, E3 +473899.464}
SPL {X  -164.446, Y  +358.564, Z    +0.000, E1   +15.149, E3 +473864.675}
SPL {X  -165.379, Y  +369.025, Z    +0.000, E1    +9.158, E3 +473870.400}
SPL {X  -165.612, Y  +374.969, Z    +0.000, E1    +5.630, E3 +473873.075}
SPL {X  -165.650, Y  +383.362, Z    +0.000, E1    +0.177, E3 +473857.694}
SPL {X  -165.650, Y  +383.923, Z    +0.000, E1    -0.215, E3 +473870.851}
SPL {X  -165.650, Y  +388.083, Z    +0.000, E1    -3.355, E3 +473869.715}
SPL {X  -165.650, Y  +393.983, Z    +0.000, E1    -8.501, E3 +473866.113}
SPL {X  -165.650, Y  +402.241, Z    +0.000, E1   -16.711, E3 +473860.625}
SPL {X  -165.650, Y  +416.345, Z    +0.000, E1   -29.511, E3 +473860.417}
SPL {X  -165.650, Y  +422.331, Z    +0.000, E1   -27.760, E3 +473885.916}
SPL {X  -165.650, Y  +441.276, Z    +0.000, E1   -37.343, E3 +473895.773}
SPL {X  -165.650, Y  +462.890, Z    +0.000, E1   -40.484, E3 +473929.856}
ENDSPLINE

SPLINE
SPL {X  -165.650, Y  +446.920, Z    +0.000, E1   -31.238, E3 +473942.182}
ENDSPLINE

SPLINE
SPL {X  -165.650, Y  +447.935, Z    +0.000, E1   -30.213, E3 +473952.470}
SPL {X  -165.650, Y  +451.020, Z    +0.000, E1   -30.224, E3 +473963.290}
SPL {X  -165.650, Y  +454.519, Z    +0.000, E1   -30.374, E3 +473974.472}
SPL {X  -165.650, Y  +456.542, Z    +0.000, E1   -29.986, E3 +473984.217}
SPL {X  -165.650, Y  +460.618, Z    +0.000, E1   -30.298, E3 +473996.537}
SPL {X  -165.650, Y  +463.853, Z    +0.000, E1   -30.103, E3 +474009.138}
SPL {X  -165.650, Y  +467.246, Z    +0.000, E1   -30.279, E3 +474019.868}
SPL {X  -165.650, Y  +469.780, Z    +0.000, E1   -30.237, E3 +474028.994}
SPL {X  -165.650, Y  +472.566, Z    +0.000, E1   -30.124, E3 +474039.651}
SPL {X  -165.650, Y  +476.540, Z    +0.000, E1   -30.193, E3 +474053.195}
SPL {X  -165.650, Y  +480.320, Z    +0.000, E1   -30.163, E3 +474066.673}
SPL {X  -165.650, Y  +484.477, Z    +0.000, E1   -30.274, E3 +474080.563}
SPL {X  -165.650, Y  +488.041, Z    +0.000, E1   -30.253, E3 +474093.118}
SPL {X  -165.650, Y  +491.281, Z    +0.000, E1   -30.148, E3 +474105.256}
SPL {X  -165.650, Y  +495.051, Z    +0.000, E1   -30.213, E3 +474118.064}
SPL {X  -165.650, Y  +498.418, Z    +0.000, E1   -30.282, E3 +474129.357}
SPL {X  -165.650, Y  +500.833, Z    +0.000, E1   -30.191, E3 +474138.406}
SPL {X  -165.650, Y  +504.246, Z    +0.000, E1   -30.231, E3 +474150.272}
SPL {X  -165.650, Y  +507.017, Z    +0.000, E1   -30.108, E3 +474160.681}
SPL {X  -165.650, Y  +510.660, Z    +0.000, E1   -30.223, E3 +474172.948}
SPL {X  -165.650, Y  +515.918, Z    +0.000, E1   -30.316, E3 +474190.756}
SPL {X  -165.650, Y  +520.621, Z    +0.000, E1   -30.198, E3 +474208.041}
SPL {X  -165.650, Y  +525.344, Z    +0.000, E1   -30.269, E3 +474224.098}
SPL {X  -165.650, Y  +528.152, Z    +0.000, E1   -29.991, E3 +474235.739}
SPL {X  -165.650, Y  +531.783, Z    +0.000, E1   -30.416, E3 +474245.632}
SPL {X  -165.650, Y  +534.115, Z    +0.000, E1   -30.089, E3 +474256.014}
SPL {X  -165.650, Y  +538.363, Z    +0.000, E1   -30.232, E3 +474270.184}
SPL {X  -165.650, Y  +543.650, Z    +0.000, E1   -30.281, E3 +474288.403}
SPL {X  -165.650, Y  +547.199, Z    +0.000, E1   -30.132, E3 +474301.662}
SPL {X  -165.650, Y  +550.512, Z    +0.000, E1   -30.197, E3 +474312.988}
SPL {X  -165.650, Y  +554.908, Z    +0.000, E1   -30.180, E3 +474328.649}
SPL {X  -165.650, Y  +560.243, Z    +0.000, E1   -30.214, E3 +474347.275}
SPL {X  -165.650, Y  +565.528, Z    +0.000, E1   -30.192, E3 +474365.967}
SPL {X  -165.650, Y  +570.048, Z    +0.000, E1   -30.238, E3 +474381.399}
SPL {X  -165.650, Y  +573.110, Z    +0.000, E1   -30.057, E3 +474393.384}
SPL {X  -165.650, Y  +577.587, Z    +0.000, E1   -30.270, E3 +474407.822}
SPL {X  -165.650, Y  +581.190, Z    +0.000, E1   -30.107, E3 +474421.462}
SPL {X  -165.650, Y  +585.053, Z    +0.000, E1   -30.090, E3 +474435.332}
ENDSPLINE

SPLINE
SPL {X  -165.650, Y  +484.445, Z    +0.000, E1   +32.277, E3 +474452.736}
SPL {X  -165.650, Y  +481.524, Z    +0.000, E1   +31.089, E3 +474470.187}
SPL {X  -165.650, Y  +478.014, Z    +0.000, E1   +30.826, E3 +474483.795}
SPL {X  -165.650, Y  +474.473, Z    +0.000, E1   +30.943, E3 +474495.119}
SPL {X  -165.650, Y  +471.826, Z    +0.000, E1   +30.770, E3 +474505.303}
SPL {X  -165.650, Y  +467.753, Z    +0.000, E1   +30.878, E3 +474518.676}
SPL {X  -165.650, Y  +463.837, Z    +0.000, E1   +30.924, E3 +474531.610}
SPL {X  -165.650, Y  +461.106, Z    +0.000, E1   +30.916, E3 +474540.997}
SPL {X  -165.650, Y  +457.156, Z    +0.000, E1   +30.860, E3 +474555.073}
SPL {X  -165.650, Y  +453.156, Z    +0.000, E1   +30.934, E3 +474568.047}
SPL {X  -165.650, Y  +450.433, Z    +0.000, E1   +30.789, E3 +474578.403}
SPL {X  -165.650, Y  +447.097, Z    +0.000, E1   +30.843, E3 +474589.451}
SPL {X  -165.650, Y  +443.673, Z    +0.000, E1   +30.907, E3 +474600.759}
SPL {X  -165.650, Y  +439.486, Z    +0.000, E1   +30.857, E3 +474615.568}
SPL {X  -165.650, Y  +434.043, Z    +0.000, E1   +30.950, E3 +474633.584}
SPL {X  -165.650, Y  +430.419, Z    +0.000, E1   +30.895, E3 +474646.087}
SPL {X  -165.650, Y  +427.340, Z    +0.000, E1   +30.870, E3 +474656.914}
SPL {X  -165.650, Y  +422.641, Z    +0.000, E1   +30.884, E3 +474673.003}
SPL {X  -165.650, Y  +417.366, Z    +0.000, E1   +30.879, E3 +474691.109}
SPL {X  -165.650, Y  +412.139, Z    +0.000, E1   +30.870, E3 +474709.058}
SPL {X  -165.650, Y  +406.834, Z    +0.000, E1   +30.919, E3 +474726.887}
SPL {X  -165.650, Y  +402.516, Z    +0.000, E1   +30.874, E3 +474741.809}
SPL {X  -165.650, Y  +398.147, Z    +0.000, E1   +30.902, E3 +474756.688}
SPL {X  -165.650, Y  +394.694, Z    +0.000, E1   +30.805, E3 +474768.996}
SPL {X  -165.650, Y  +391.522, Z    +0.000, E1   +30.837, E3 +474779.677}
SPL {X  -165.650, Y  +387.533, Z    +0.000, E1   +30.858, E3 +474793.303}
SPL {X  -165.650, Y  +383.627, Z    +0.000, E1   +30.885, E3 +474806.363}
SPL {X  -165.650, Y  +380.752, Z    +0.000, E1   +30.927, E3 +474815.877}
SPL {X  -165.648, Y  +377.739, Z    +0.000, E1   +30.835, E3 +474826.887}
SPL {X  -165.594, Y  +374.183, Z    +0.000, E1   +30.878, E3 +474838.723}
SPL {X  -165.492, Y  +371.263, Z    +0.000, E1   +30.913, E3 +474848.418}
SPL {X  -165.379, Y  +369.027, Z    +0.000, E1   +30.727, E3 +474857.357}
SPL {X  -165.167, Y  +365.866, Z    +0.000, E1   +30.741, E3 +474868.131}
SPL {X  -164.892, Y  +362.671, Z    +0.000, E1   +30.830, E3 +474878.455}
SPL {X  -164.570, Y  +359.612, Z    +0.000, E1   +30.773, E3 +474889.268}
SPL {X  -164.104, Y  +355.923, Z    +0.000, E1   +30.626, E3 +474902.984}
SPL {X  -163.573, Y  +352.353, Z    +0.000, E1   +30.451, E3 +474916.249}
SPL {X  -162.476, Y  +346.230, Z    +0.000, E1   +31.677, E3 +474928.830}
SPL {X  -152.976, Y  +314.952, Z    +0.000, E1   +38.607, E3 +474977.795}
SPL {X  -137.967, Y  +286.821, Z    +0.000, E1   +43.969, E3 +475021.016}
ENDSPLINE

SPLINE
SPL {X  -153.316, Y  +315.777, Z    +0.000, E1   +33.140, E3 +475063.644}
SPL {X  -164.446, Y  +358.564, Z    +0.000, E1   +15.149, E3 +475028.854}
SPL {X  -165.379, Y  +369.025, Z    +0.000, E1    +9.158, E3 +475034.579}
SPL {X  -165.612, Y  +374.969, Z    +0.000, E1    +5.630, E3 +475037.255}
SPL {X  -165.650, Y  +383.362, Z    +0.000, E1    +0.177, E3 +475021.873}
SPL {X  -165.650, Y  +383.923, Z    +0.000, E1    -0.215, E3 +475035.030}
SPL {X  -165.650, Y  +388.083, Z    +0.000, E1    -3.355, E3 +475033.894}
SPL {X  -165.650, Y  +393.983, Z    +0.000, E1    -8.501, E3 +475030.292}
SPL {X  -165.650, Y  +402.241, Z    +0.000, E1   -16.711, E3 +475024.804}
SPL {X  -165.650, Y  +416.345, Z    +0.000, E1   -29.511, E3 +475024.596}
SPL {X  -165.650, Y  +422.331, Z    +0.000, E1   -27.760, E3 +475050.095}
SPL {X  -165.650, Y  +441.276, Z    +0.000, E1   -37.343, E3 +475059.952}
SPL {X  -165.650, Y  +462.890, Z    +0.000, E1   -40.484, E3 +475094.035}
ENDSPLINE

SPLINE
SPL {X  -165.650, Y  +446.920, Z    +0.000, E1   -31.238, E3 +475106.361}
ENDSPLINE

SPLINE
SPL {X  -165.650, Y  +447.935, Z    +0.000, E1   -30.213, E3 +475116.649}
SPL {X  -165.650, Y  +451.020, Z    +0.000, E1   -30.224, E3 +475127.469}
SPL {X  -165.650, Y  +454.519, Z    +0.000, E1   -30.374, E3 +475138.651}
SPL {X  -165.650, Y  +457.429, Z    +0.000, E1   -30.029, E3 +475151.353}
SPL {X  -165.650, Y  +461.678, Z    +0.000, E1   -30.426, E3 +475163.478}
SPL {X  -165.650, Y  +463.853, Z    +0.000, E1   -30.103, E3 +475173.317}
SPL {X  -165.650, Y  +468.397, Z    +0.000, E1   -30.302, E3 +475188.121}
SPL {X  -165.650, Y  +472.566, Z    +0.000, E1   -30.124, E3 +475203.831}
SPL {X  -165.650, Y  +476.540, Z    +0.000, E1   -30.193, E3 +475217.375}
SPL {X  -165.650, Y  +481.042, Z    +0.000, E1   -30.192, E3 +475233.320}
SPL {X  -165.650, Y  +485.236, Z    +0.000, E1   -30.294, E3 +475247.175}
SPL {X  -165.650, Y  +489.057, Z    +0.000, E1   -30.341, E3 +475260.381}
SPL {X  -165.650, Y  +491.647, Z    +0.000, E1   -29.894, E3 +475272.315}
SPL {X  -165.650, Y  +495.051, Z    +0.000, E1   -30.213, E3 +475282.244}
SPL {X  -165.650, Y  +498.418, Z    +0.000, E1   -30.282, E3 +475293.536}
SPL {X  -165.650, Y  +502.421, Z    +0.000, E1   -30.263, E3 +475307.894}
SPL {X  -165.650, Y  +506.344, Z    +0.000, E1   -30.129, E3 +475322.423}
SPL {X  -165.650, Y  +509.866, Z    +0.000, E1   -30.236, E3 +475334.093}
SPL {X  -165.650, Y  +513.685, Z    +0.000, E1   -30.234, E3 +475347.589}
SPL {X  -165.650, Y  +517.919, Z    +0.000, E1   -30.227, E3 +475362.496}
SPL {X  -165.650, Y  +521.521, Z    +0.000, E1   -30.210, E3 +475375.171}
SPL {X  -165.650, Y  +525.344, Z    +0.000, E1   -30.269, E3 +475388.277}
SPL {X  -165.650, Y  +528.152, Z    +0.000, E1   -29.991, E3 +475399.918}
SPL {X  -165.650, Y  +531.783, Z    +0.000, E1   -30.416, E3 +475409.811}
SPL {X  -165.650, Y  +534.115, Z    +0.000, E1   -30.089, E3 +475420.193}
SPL {X  -165.650, Y  +537.522, Z    +0.000, E1   -30.251, E3 +475431.107}
SPL {X  -165.650, Y  +540.621, Z    +0.000, E1   -30.014, E3 +475443.668}
SPL {X  -165.650, Y  +544.944, Z    +0.000, E1   -30.447, E3 +475455.868}
SPL {X  -165.650, Y  +548.549, Z    +0.000, E1   -30.216, E3 +475470.191}
SPL {X  -165.650, Y  +553.092, Z    +0.000, E1   -30.157, E3 +475486.534}
SPL {X  -165.650, Y  +556.274, Z    +0.000, E1   -30.127, E3 +475497.788}
SPL {X  -165.650, Y  +560.243, Z    +0.000, E1   -30.214, E3 +475511.454}
SPL {X  -165.650, Y  +565.528, Z    +0.000, E1   -30.192, E3 +475530.147}
SPL {X  -165.650, Y  +570.048, Z    +0.000, E1   -30.238, E3 +475545.578}
SPL {X  -165.650, Y  +573.110, Z    +0.000, E1   -30.057, E3 +475557.563}
SPL {X  -165.650, Y  +577.587, Z    +0.000, E1   -30.270, E3 +475572.002}
SPL {X  -165.650, Y  +581.190, Z    +0.000, E1   -30.107, E3 +475585.641}
SPL {X  -165.650, Y  +585.053, Z    +0.000, E1   -30.090, E3 +475599.511}
ENDSPLINE

SPLINE
SPL {X  -165.650, Y  +484.445, Z    +0.000, E1   +32.277, E3 +475616.916}
SPL {X  -165.650, Y  +481.524, Z    +0.000, E1   +31.089, E3 +475634.366}
SPL {X  -165.650, Y  +478.014, Z    +0.000, E1   +30.826, E3 +475647.974}
SPL {X  -165.650, Y  +474.473, Z    +0.000, E1   +30.943, E3 +475659.298}
SPL {X  -165.650, Y  +471.826, Z    +0.000, E1   +30.770, E3 +475669.482}
SPL {X  -165.650, Y  +467.753, Z    +0.000, E1   +30.878, E3 +475682.855}
SPL {X  -165.650, Y  +463.837, Z    +0.000, E1   +30.924, E3 +475695.789}
SPL {X  -165.650, Y  +461.106, Z    +0.000, E1   +30.916, E3 +475705.176}
SPL {X  -165.650, Y  +458.435, Z    +0.000, E1   +30.759, E3 +475715.384}
SPL {X  -165.650, Y  +454.220, Z    +0.000, E1   +30.954, E3 +475728.617}
SPL {X  -165.650, Y  +450.433, Z    +0.000, E1   +30.789, E3 +475742.582}
SPL {X  -165.650, Y  +447.097, Z    +0.000, E1   +30.843, E3 +475753.630}
SPL {X  -165.650, Y  +443.673, Z    +0.000, E1   +30.907, E3 +475764.938}
SPL {X  -165.650, Y  +440.976, Z    +0.000, E1   +30.719, E3 +475775.395}
SPL {X  -165.650, Y  +436.324, Z    +0.000, E1   +30.994, E3 +475789.681}
SPL {X  -165.650, Y  +432.765, Z    +0.000, E1   +30.831, E3 +475802.681}
SPL {X  -165.650, Y  +429.309, Z    +0.000, E1   +30.920, E3 +475814.022}
SPL {X  -165.650, Y  +424.918, Z    +0.000, E1   +30.862, E3 +475829.479}
SPL {X  -165.650, Y  +421.437, Z    +0.000, E1   +30.833, E3 +475841.447}
SPL {X  -165.650, Y  +417.366, Z    +0.000, E1   +30.879, E3 +475855.288}
SPL {X  -165.650, Y  +413.181, Z    +0.000, E1   +30.815, E3 +475869.885}
SPL {X  -165.650, Y  +408.547, Z    +0.000, E1   +30.964, E3 +475884.888}
SPL {X  -165.650, Y  +403.421, Z    +0.000, E1   +30.863, E3 +475903.106}
SPL {X  -165.650, Y  +398.147, Z    +0.000, E1   +30.902, E3 +475920.867}
SPL {X  -165.650, Y  +394.694, Z    +0.000, E1   +30.805, E3 +475933.175}
SPL {X  -165.650, Y  +391.522, Z    +0.000, E1   +30.837, E3 +475943.856}
SPL {X  -165.650, Y  +387.533, Z    +0.000, E1   +30.858, E3 +475957.482}
SPL {X  -165.650, Y  +383.627, Z    +0.000, E1   +30.885, E3 +475970.542}
SPL {X  -165.650, Y  +379.886, Z    +0.000, E1   +30.887, E3 +475983.430}
SPL {X  -165.614, Y  +375.058, Z    +0.000, E1   +30.905, E3 +475999.884}
SPL {X  -165.492, Y  +371.263, Z    +0.000, E1   +30.913, E3 +476012.597}
SPL {X  -165.379, Y  +369.027, Z    +0.000, E1   +30.727, E3 +476021.536}
SPL {X  -165.167, Y  +365.866, Z    +0.000, E1   +30.741, E3 +476032.310}
SPL {X  -164.892, Y  +362.671, Z    +0.000, E1   +30.830, E3 +476042.634}
SPL {X  -164.570, Y  +359.612, Z    +0.000, E1   +30.773, E3 +476053.447}
SPL {X  -164.104, Y  +355.923, Z    +0.000, E1   +30.626, E3 +476067.163}
SPL {X  -163.573, Y  +352.353, Z    +0.000, E1   +30.451, E3 +476080.428}
SPL {X  -162.476, Y  +346.230, Z    +0.000, E1   +31.677, E3 +476093.009}
SPL {X  -152.976, Y  +314.952, Z    +0.000, E1   +38.607, E3 +476141.974}
SPL {X  -137.967, Y  +286.821, Z    +0.000, E1   +43.969, E3 +476185.195}
ENDSPLINE

SPLINE
SPL {X  -153.316, Y  +315.777, Z    +0.000, E1   +33.140, E3 +476227.823}
SPL {X  -164.446, Y  +358.564, Z    +0.000, E1   +15.149, E3 +476193.033}
SPL {X  -165.510, Y  +371.680, Z    +0.000, E1    +7.684, E3 +476197.089}
SPL {X  -165.628, Y  +375.818, Z    +0.000, E1    +5.016, E3 +476205.018}
SPL {X  -165.650, Y  +383.362, Z    +0.000, E1    +0.177, E3 +476186.052}
SPL {X  -165.650, Y  +383.923, Z    +0.000, E1    -0.215, E3 +476199.209}
SPL {X  -165.650, Y  +388.083, Z    +0.000, E1    -3.355, E3 +476198.073}
SPL {X  -165.650, Y  +393.983, Z    +0.000, E1    -8.501, E3 +476194.471}
SPL {X  -165.650, Y  +402.241, Z    +0.000, E1   -16.711, E3 +476188.983}
SPL {X  -165.650, Y  +414.811, Z    +0.000, E1   -28.314, E3 +476188.513}
SPL {X  -165.650, Y  +423.479, Z    +0.000, E1   -29.012, E3 +476212.442}
SPL {X  -165.650, Y  +441.276, Z    +0.000, E1   -37.343, E3 +476224.131}
SPL {X  -165.650, Y  +462.890, Z    +0.000, E1   -40.484, E3 +476258.214}
ENDSPLINE

SPLINE
SPL {X  -165.650, Y  +446.920, Z    +0.000, E1   -31.238, E3 +476270.540}
ENDSPLINE

SPLINE
SPL {X  -165.650, Y  +447.935, Z    +0.000, E1   -30.213, E3 +476280.828}
SPL {X  -165.650, Y  +451.020, Z    +0.000, E1   -30.224, E3 +476291.648}
SPL {X  -165.650, Y  +454.519, Z    +0.000, E1   -30.374, E3 +476302.830}
SPL {X  -165.650, Y  +456.542, Z    +0.000, E1   -29.986, E3 +476312.575}
SPL {X  -165.650, Y  +460.618, Z    +0.000, E1   -30.298, E3 +476324.896}
SPL {X  -165.650, Y  +463.853, Z    +0.000, E1   -30.103, E3 +476337.496}
SPL {X  -165.650, Y  +468.397, Z    +0.000, E1   -30.302, E3 +476352.300}
SPL {X  -165.650, Y  +472.566, Z    +0.000, E1   -30.124, E3 +476368.010}
SPL {X  -165.650, Y  +475.265, Z    +0.000, E1   -30.034, E3 +476378.047}
SPL {X  -165.650, Y  +477.862, Z    +0.000, E1   -30.319, E3 +476385.239}
SPL {X  -165.650, Y  +481.042, Z    +0.000, E1   -30.192, E3 +476397.499}
SPL {X  -165.650, Y  +485.236, Z    +0.000, E1   -30.294, E3 +476411.354}
SPL {X  -165.650, Y  +488.041, Z    +0.000, E1   -30.253, E3 +476421.476}
SPL {X  -165.650, Y  +491.281, Z    +0.000, E1   -30.148, E3 +476433.614}
SPL {X  -165.650, Y  +495.051, Z    +0.000, E1   -30.213, E3 +476446.423}
SPL {X  -165.650, Y  +499.546, Z    +0.000, E1   -30.283, E3 +476461.865}
SPL {X  -165.650, Y  +503.544, Z    +0.000, E1   -30.247, E3 +476475.934}
SPL {X  -165.650, Y  +506.344, Z    +0.000, E1   -30.129, E3 +476486.603}
SPL {X  -165.650, Y  +510.660, Z    +0.000, E1   -30.223, E3 +476501.306}
SPL {X  -165.650, Y  +514.670, Z    +0.000, E1   -30.278, E3 +476514.816}
SPL {X  -165.650, Y  +517.919, Z    +0.000, E1   -30.227, E3 +476526.675}
SPL {X  -165.650, Y  +521.521, Z    +0.000, E1   -30.210, E3 +476539.350}
SPL {X  -165.650, Y  +525.344, Z    +0.000, E1   -30.269, E3 +476552.456}
SPL {X  -165.650, Y  +528.152, Z    +0.000, E1   -29.991, E3 +476564.097}
SPL {X  -165.650, Y  +531.783, Z    +0.000, E1   -30.416, E3 +476573.990}
SPL {X  -165.650, Y  +534.115, Z    +0.000, E1   -30.089, E3 +476584.372}
SPL {X  -165.650, Y  +537.522, Z    +0.000, E1   -30.251, E3 +476595.286}
SPL {X  -165.650, Y  +540.621, Z    +0.000, E1   -30.014, E3 +476607.847}
SPL {X  -165.650, Y  +544.944, Z    +0.000, E1   -30.447, E3 +476620.047}
SPL {X  -165.650, Y  +547.199, Z    +0.000, E1   -30.132, E3 +476630.020}
SPL {X  -165.650, Y  +550.512, Z    +0.000, E1   -30.197, E3 +476641.346}
SPL {X  -165.650, Y  +553.852, Z    +0.000, E1   -30.156, E3 +476653.287}
SPL {X  -165.650, Y  +557.277, Z    +0.000, E1   -30.150, E3 +476665.461}
SPL {X  -165.650, Y  +561.168, Z    +0.000, E1   -30.194, E3 +476678.843}
SPL {X  -165.650, Y  +564.449, Z    +0.000, E1   -30.167, E3 +476690.526}
SPL {X  -165.650, Y  +566.935, Z    +0.000, E1   -30.135, E3 +476699.432}
SPL {X  -165.650, Y  +570.048, Z    +0.000, E1   -30.238, E3 +476709.757}
SPL {X  -165.650, Y  +573.110, Z    +0.000, E1   -30.057, E3 +476721.742}
SPL {X  -165.650, Y  +577.587, Z    +0.000, E1   -30.270, E3 +476736.181}
SPL {X  -165.650, Y  +581.190, Z    +0.000, E1   -30.107, E3 +476749.820}
SPL {X  -165.650, Y  +585.053, Z    +0.000, E1   -30.090, E3 +476763.690}
ENDSPLINE

SPLINE
SPL {X  -165.650, Y  +484.445, Z    +0.000, E1   +32.277, E3 +476781.095}
SPL {X  -165.650, Y  +481.524, Z    +0.000, E1   +31.089, E3 +476798.545}
SPL {X  -165.650, Y  +478.014, Z    +0.000, E1   +30.826, E3 +476812.153}
SPL {X  -165.650, Y  +474.473, Z    +0.000, E1   +30.943, E3 +476823.477}
SPL {X  -165.650, Y  +471.826, Z    +0.000, E1   +30.770, E3 +476833.661}
SPL {X  -165.650, Y  +467.753, Z    +0.000, E1   +30.878, E3 +476847.034}
SPL {X  -165.650, Y  +463.837, Z    +0.000, E1   +30.924, E3 +476859.968}
SPL {X  -165.650, Y  +461.106, Z    +0.000, E1   +30.916, E3 +476869.355}
SPL {X  -165.650, Y  +458.435, Z    +0.000, E1   +30.759, E3 +476879.563}
SPL {X  -165.650, Y  +454.220, Z    +0.000, E1   +30.954, E3 +476892.796}
SPL {X  -165.650, Y  +450.433, Z    +0.000, E1   +30.789, E3 +476906.761}
SPL {X  -165.650, Y  +447.097, Z    +0.000, E1   +30.843, E3 +476917.809}
SPL {X  -165.650, Y  +443.673, Z    +0.000, E1   +30.907, E3 +476929.117}
SPL {X  -165.650, Y  +440.976, Z    +0.000, E1   +30.719, E3 +476939.574}
SPL {X  -165.650, Y  +437.973, Z    +0.000, E1   +30.928, E3 +476948.446}
SPL {X  -165.650, Y  +434.043, Z    +0.000, E1   +30.950, E3 +476961.942}
SPL {X  -165.650, Y  +430.419, Z    +0.000, E1   +30.895, E3 +476974.445}
SPL {X  -165.650, Y  +427.340, Z    +0.000, E1   +30.870, E3 +476985.272}
SPL {X  -165.650, Y  +422.641, Z    +0.000, E1   +30.884, E3 +477001.361}
SPL {X  -165.650, Y  +418.489, Z    +0.000, E1   +30.835, E3 +477015.743}
SPL {X  -165.650, Y  +414.127, Z    +0.000, E1   +30.869, E3 +477030.652}
SPL {X  -165.650, Y  +408.547, Z    +0.000, E1   +30.964, E3 +477049.067}
SPL {X  -165.650, Y  +405.433, Z    +0.000, E1   +30.730, E3 +477061.044}
SPL {X  -165.650, Y  +402.516, Z    +0.000, E1   +30.874, E3 +477070.167}
SPL {X  -165.650, Y  +398.147, Z    +0.000, E1   +30.902, E3 +477085.046}
SPL {X  -165.650, Y  +394.694, Z    +0.000, E1   +30.805, E3 +477097.354}
SPL {X  -165.650, Y  +391.522, Z    +0.000, E1   +30.837, E3 +477108.035}
SPL {X  -165.650, Y  +387.533, Z    +0.000, E1   +30.858, E3 +477121.661}
SPL {X  -165.650, Y  +383.627, Z    +0.000, E1   +30.885, E3 +477134.721}
SPL {X  -165.650, Y  +379.886, Z    +0.000, E1   +30.887, E3 +477147.610}
SPL {X  -165.614, Y  +375.058, Z    +0.000, E1   +30.905, E3 +477164.063}
SPL {X  -165.492, Y  +371.263, Z    +0.000, E1   +30.913, E3 +477176.777}
SPL {X  -165.379, Y  +369.027, Z    +0.000, E1   +30.727, E3 +477185.715}
SPL {X  -165.167, Y  +365.866, Z    +0.000, E1   +30.741, E3 +477196.489}
SPL {X  -164.892, Y  +362.671, Z    +0.000, E1   +30.830, E3 +477206.813}
SPL {X  -164.570, Y  +359.612, Z    +0.000, E1   +30.773, E3 +477217.626}
SPL {X  -164.104, Y  +355.923, Z    +0.000, E1   +30.626, E3 +477231.342}
SPL {X  -163.573, Y  +352.353, Z    +0.000, E1   +30.451, E3 +477244.607}
SPL {X  -162.976, Y  +348.856, Z    +0.000, E1   +30.757, E3 +477254.531}
SPL {X  -161.497, Y  +341.640, Z    +0.000, E1   +33.276, E3 +477261.808}
SPL {X  -152.976, Y  +314.952, Z    +0.000, E1   +38.607, E3 +477306.153}
SPL {X  -137.967, Y  +286.821, Z    +0.000, E1   +43.969, E3 +477349.374}
ENDSPLINE

SPLINE
SPL {X  -149.143, Y  +306.414, Z    +0.000, E1   +36.361, E3 +477400.507}
SPL {X  -164.268, Y  +357.145, Z    +0.000, E1   +15.880, E3 +477358.266}
SPL {X  -165.379, Y  +369.025, Z    +0.000, E1    +9.158, E3 +477362.937}
SPL {X  -165.612, Y  +374.969, Z    +0.000, E1    +5.630, E3 +477365.613}
SPL {X  -165.650, Y  +383.362, Z    +0.000, E1    +0.177, E3 +477350.231}
SPL {X  -165.650, Y  +383.923, Z    +0.000, E1    -0.215, E3 +477363.389}
SPL {X  -165.650, Y  +388.083, Z    +0.000, E1    -3.355, E3 +477362.252}
SPL {X  -165.650, Y  +393.983, Z    +0.000, E1    -8.501, E3 +477358.650}
SPL {X  -165.650, Y  +402.241, Z    +0.000, E1   -16.711, E3 +477353.162}
SPL {X  -165.650, Y  +416.345, Z    +0.000, E1   -29.511, E3 +477352.954}
SPL {X  -165.650, Y  +422.331, Z    +0.000, E1   -27.760, E3 +477378.453}
SPL {X  -165.650, Y  +441.276, Z    +0.000, E1   -37.343, E3 +477388.310}
SPL {X  -165.650, Y  +462.890, Z    +0.000, E1   -40.484, E3 +477422.393}
ENDSPLINE

SPLINE
SPL {X  -165.650, Y  +446.920, Z    +0.000, E1   -31.238, E3 +477434.719}
ENDSPLINE

SPLINE
SPL {X  -165.650, Y  +447.935, Z    +0.000, E1   -30.213, E3 +477445.007}
SPL {X  -165.650, Y  +451.020, Z    +0.000, E1   -30.224, E3 +477455.827}
SPL {X  -165.650, Y  +454.519, Z    +0.000, E1   -30.374, E3 +477467.010}
SPL {X  -165.650, Y  +456.542, Z    +0.000, E1   -29.986, E3 +477476.754}
SPL {X  -165.650, Y  +460.618, Z    +0.000, E1   -30.298, E3 +477489.075}
SPL {X  -165.650, Y  +463.853, Z    +0.000, E1   -30.103, E3 +477501.676}
SPL {X  -165.650, Y  +468.397, Z    +0.000, E1   -30.302, E3 +477516.479}
SPL {X  -165.650, Y  +472.566, Z    +0.000, E1   -30.124, E3 +477532.189}
SPL {X  -165.650, Y  +476.540, Z    +0.000, E1   -30.193, E3 +477545.733}
SPL {X  -165.650, Y  +480.320, Z    +0.000, E1   -30.163, E3 +477559.211}
SPL {X  -165.650, Y  +484.477, Z    +0.000, E1   -30.274, E3 +477573.100}
SPL {X  -165.650, Y  +488.041, Z    +0.000, E1   -30.253, E3 +477585.655}
SPL {X  -165.650, Y  +491.281, Z    +0.000, E1   -30.148, E3 +477597.793}
SPL {X  -165.650, Y  +495.051, Z    +0.000, E1   -30.213, E3 +477610.602}
SPL {X  -165.650, Y  +499.546, Z    +0.000, E1   -30.283, E3 +477626.045}
SPL {X  -165.650, Y  +503.544, Z    +0.000, E1   -30.247, E3 +477640.113}
SPL {X  -165.650, Y  +506.344, Z    +0.000, E1   -30.129, E3 +477650.782}
SPL {X  -165.650, Y  +509.866, Z    +0.000, E1   -30.236, E3 +477662.451}
SPL {X  -165.650, Y  +513.685, Z    +0.000, E1   -30.234, E3 +477675.947}
SPL {X  -165.650, Y  +517.919, Z    +0.000, E1   -30.227, E3 +477690.854}
SPL {X  -165.650, Y  +521.521, Z    +0.000, E1   -30.210, E3 +477703.529}
SPL {X  -165.650, Y  +525.344, Z    +0.000, E1   -30.269, E3 +477716.635}
SPL {X  -165.650, Y  +528.152, Z    +0.000, E1   -29.991, E3 +477728.276}
SPL {X  -165.650, Y  +531.783, Z    +0.000, E1   -30.416, E3 +477738.169}
SPL {X  -165.650, Y  +534.115, Z    +0.000, E1   -30.089, E3 +477748.551}
SPL {X  -165.650, Y  +537.522, Z    +0.000, E1   -30.251, E3 +477759.465}
SPL {X  -165.650, Y  +540.621, Z    +0.000, E1   -30.014, E3 +477772.026}
SPL {X  -165.650, Y  +544.944, Z    +0.000, E1   -30.447, E3 +477784.226}
SPL {X  -165.650, Y  +547.199, Z    +0.000, E1   -30.132, E3 +477794.199}
SPL {X  -165.650, Y  +550.512, Z    +0.000, E1   -30.197, E3 +477805.525}
SPL {X  -165.650, Y  +553.852, Z    +0.000, E1   -30.156, E3 +477817.466}
SPL {X  -165.650, Y  +557.277, Z    +0.000, E1   -30.150, E3 +477829.640}
SPL {X  -165.650, Y  +561.168, Z    +0.000, E1   -30.194, E3 +477843.022}
SPL {X  -165.650, Y  +565.528, Z    +0.000, E1   -30.192, E3 +477858.505}
SPL {X  -165.650, Y  +570.048, Z    +0.000, E1   -30.238, E3 +477873.936}
SPL {X  -165.650, Y  +573.110, Z    +0.000, E1   -30.057, E3 +477885.921}
SPL {X  -165.650, Y  +577.587, Z    +0.000, E1   -30.270, E3 +477900.360}
SPL {X  -165.650, Y  +581.190, Z    +0.000, E1   -30.107, E3 +477913.999}
SPL {X  -165.650, Y  +585.053, Z    +0.000, E1   -30.090, E3 +477927.869}
ENDSPLINE

SPLINE
SPL {X  -165.650, Y  +484.445, Z    +0.000, E1   +32.277, E3 +477945.274}
SPL {X  -165.650, Y  +481.524, Z    +0.000, E1   +31.089, E3 +477962.724}
SPL {X  -165.650, Y  +478.014, Z    +0.000, E1   +30.826, E3 +477976.332}
SPL {X  -165.650, Y  +474.473, Z    +0.000, E1   +30.943, E3 +477987.656}
SPL {X  -165.650, Y  +471.826, Z    +0.000, E1   +30.770, E3 +477997.840}
SPL {X  -165.650, Y  +467.753, Z    +0.000, E1   +30.878, E3 +478011.213}
SPL {X  -165.650, Y  +463.837, Z    +0.000, E1   +30.924, E3 +478024.147}
SPL {X  -165.650, Y  +461.106, Z    +0.000, E1   +30.916, E3 +478033.534}
SPL {X  -165.650, Y  +457.156, Z    +0.000, E1   +30.860, E3 +478047.611}
SPL {X  -165.650, Y  +453.156, Z    +0.000, E1   +30.934, E3 +478060.585}
SPL {X  -165.650, Y  +450.433, Z    +0.000, E1   +30.789, E3 +478070.940}
SPL {X  -165.650, Y  +447.097, Z    +0.000, E1   +30.843, E3 +478081.989}
SPL {X  -165.650, Y  +443.673, Z    +0.000, E1   +30.907, E3 +478093.296}
SPL {X  -165.650, Y  +439.486, Z    +0.000, E1   +30.857, E3 +478108.105}
SPL {X  -165.650, Y  +435.146, Z    +0.000, E1   +30.969, E3 +478122.025}
SPL {X  -165.650, Y  +432.765, Z    +0.000, E1   +30.831, E3 +478131.039}
SPL {X  -165.650, Y  +429.309, Z    +0.000, E1   +30.920, E3 +478142.380}
SPL {X  -165.650, Y  +424.918, Z    +0.000, E1   +30.862, E3 +478157.837}
SPL {X  -165.650, Y  +421.437, Z    +0.000, E1   +30.833, E3 +478169.806}
SPL {X  -165.650, Y  +417.366, Z    +0.000, E1   +30.879, E3 +478183.646}
SPL {X  -165.650, Y  +413.181, Z    +0.000, E1   +30.815, E3 +478198.244}
SPL {X  -165.650, Y  +408.547, Z    +0.000, E1   +30.964, E3 +478213.246}
SPL {X  -165.650, Y  +403.421, Z    +0.000, E1   +30.863, E3 +478231.464}
SPL {X  -165.650, Y  +399.681, Z    +0.000, E1   +30.933, E3 +478243.547}
SPL {X  -165.650, Y  +396.018, Z    +0.000, E1   +30.861, E3 +478256.857}
SPL {X  -165.650, Y  +391.522, Z    +0.000, E1   +30.837, E3 +478272.214}
SPL {X  -165.650, Y  +387.533, Z    +0.000, E1   +30.858, E3 +478285.840}
SPL {X  -165.650, Y  +383.627, Z    +0.000, E1   +30.885, E3 +478298.900}
SPL {X  -165.650, Y  +380.752, Z    +0.000, E1   +30.927, E3 +478308.414}
SPL {X  -165.648, Y  +377.739, Z    +0.000, E1   +30.835, E3 +478319.424}
SPL {X  -165.594, Y  +374.183, Z    +0.000, E1   +30.878, E3 +478331.261}
SPL {X  -165.429, Y  +369.945, Z    +0.000, E1   +30.850, E3 +478346.136}
SPL {X  -165.167, Y  +365.866, Z    +0.000, E1   +30.741, E3 +478360.668}
SPL {X  -164.892, Y  +362.671, Z    +0.000, E1   +30.830, E3 +478370.992}
SPL {X  -164.570, Y  +359.612, Z    +0.000, E1   +30.773, E3 +478381.805}
SPL {X  -164.287, Y  +357.291, Z    +0.000, E1   +30.513, E3 +478391.434}
SPL {X  -163.720, Y  +353.284, Z    +0.000, E1   +30.592, E3 +478404.881}
SPL {X  -162.976, Y  +348.856, Z    +0.000, E1   +30.757, E3 +478418.710}
SPL {X  -161.497, Y  +341.640, Z    +0.000, E1   +33.276, E3 +478425.988}
SPL {X  -152.976, Y  +314.952, Z    +0.000, E1   +38.607, E3 +478470.332}
SPL {X  -137.967, Y  +286.821, Z    +0.000, E1   +43.969, E3 +478513.553}
ENDSPLINE

SPLINE
SPL {X  -149.143, Y  +306.414, Z    +0.000, E1   +36.361, E3 +478564.686}
SPL {X  -164.268, Y  +357.145, Z    +0.000, E1   +15.880, E3 +478522.445}
SPL {X  -165.379, Y  +369.025, Z    +0.000, E1    +9.158, E3 +478527.116}
SPL {X  -165.612, Y  +374.969, Z    +0.000, E1    +5.630, E3 +478529.792}
SPL {X  -165.650, Y  +383.362, Z    +0.000, E1    +0.177, E3 +478514.410}
SPL {X  -165.650, Y  +383.923, Z    +0.000, E1    -0.215, E3 +478527.568}
SPL {X  -165.650, Y  +388.083, Z    +0.000, E1    -3.355, E3 +478526.431}
SPL {X  -165.650, Y  +393.983, Z    +0.000, E1    -8.501, E3 +478522.829}
SPL {X  -165.650, Y  +402.241, Z    +0.000, E1   -16.711, E3 +478517.341}
SPL {X  -165.650, Y  +416.345, Z    +0.000, E1   -29.511, E3 +478517.133}
SPL {X  -165.650, Y  +422.331, Z    +0.000, E1   -27.760, E3 +478542.632}
SPL {X  -165.650, Y  +441.276, Z    +0.000, E1   -37.343, E3 +478552.489}
SPL {X  -165.650, Y  +462.890, Z    +0.000, E1   -40.484, E3 +478586.572}
ENDSPLINE

SPLINE
SPL {X  -165.650, Y  +446.920, Z    +0.000, E1   -31.238, E3 +478598.898}
ENDSPLINE

SPLINE
SPL {X  -165.650, Y  +447.935, Z    +0.000, E1   -30.213, E3 +478609.186}
SPL {X  -165.650, Y  +451.020, Z    +0.000, E1   -30.224, E3 +478620.006}
SPL {X  -165.650, Y  +454.519, Z    +0.000, E1   -30.374, E3 +478631.189}
SPL {X  -165.650, Y  +457.429, Z    +0.000, E1   -30.029, E3 +478643.890}
SPL {X  -165.650, Y  +461.678, Z    +0.000, E1   -30.426, E3 +478656.015}
SPL {X  -165.650, Y  +463.853, Z    +0.000, E1   -30.103, E3 +478665.855}
SPL {X  -165.650, Y  +467.246, Z    +0.000, E1   -30.279, E3 +478676.585}
SPL {X  -165.650, Y  +469.780, Z    +0.000, E1   -30.237, E3 +478685.710}
SPL {X  -165.650, Y  +472.566, Z    +0.000, E1   -30.124, E3 +478696.368}
SPL {X  -165.650, Y  +475.265, Z    +0.000, E1   -30.034, E3 +478706.405}
SPL {X  -165.650, Y  +477.862, Z    +0.000, E1   -30.319, E3 +478713.597}
SPL {X  -165.650, Y  +481.042, Z    +0.000, E1   -30.192, E3 +478725.857}
SPL {X  -165.650, Y  +485.236, Z    +0.000, E1   -30.294, E3 +478739.713}
SPL {X  -165.650, Y  +488.041, Z    +0.000, E1   -30.253, E3 +478749.834}
SPL {X  -165.650, Y  +491.281, Z    +0.000, E1   -30.148, E3 +478761.972}
SPL {X  -165.650, Y  +495.051, Z    +0.000, E1   -30.213, E3 +478774.781}
SPL {X  -165.650, Y  +499.546, Z    +0.000, E1   -30.283, E3 +478790.224}
SPL {X  -165.650, Y  +503.544, Z    +0.000, E1   -30.247, E3 +478804.292}
SPL {X  -165.650, Y  +506.344, Z    +0.000, E1   -30.129, E3 +478814.961}
SPL {X  -165.650, Y  +509.866, Z    +0.000, E1   -30.236, E3 +478826.630}
SPL {X  -165.650, Y  +513.685, Z    +0.000, E1   -30.234, E3 +478840.126}
SPL {X  -165.650, Y  +517.919, Z    +0.000, E1   -30.227, E3 +478855.033}
SPL {X  -165.650, Y  +521.521, Z    +0.000, E1   -30.210, E3 +478867.708}
SPL {X  -165.650, Y  +525.344, Z    +0.000, E1   -30.269, E3 +478880.814}
SPL {X  -165.650, Y  +528.152, Z    +0.000, E1   -29.991, E3 +478892.455}
SPL {X  -165.650, Y  +531.783, Z    +0.000, E1   -30.416, E3 +478902.348}
SPL {X  -165.650, Y  +534.115, Z    +0.000, E1   -30.089, E3 +478912.730}
SPL {X  -165.650, Y  +537.522, Z    +0.000, E1   -30.251, E3 +478923.644}
SPL {X  -165.650, Y  +540.621, Z    +0.000, E1   -30.014, E3 +478936.205}
SPL {X  -165.650, Y  +544.944, Z    +0.000, E1   -30.447, E3 +478948.405}
SPL {X  -165.650, Y  +547.199, Z    +0.000, E1   -30.132, E3 +478958.379}
SPL {X  -165.650, Y  +550.512, Z    +0.000, E1   -30.197, E3 +478969.704}
SPL {X  -165.650, Y  +553.852, Z    +0.000, E1   -30.156, E3 +478981.645}
SPL {X  -165.650, Y  +557.277, Z    +0.000, E1   -30.150, E3 +478993.820}
SPL {X  -165.650, Y  +561.168, Z    +0.000, E1   -30.194, E3 +479007.201}
SPL {X  -165.650, Y  +564.449, Z    +0.000, E1   -30.167, E3 +479018.884}
SPL {X  -165.650, Y  +566.935, Z    +0.000, E1   -30.135, E3 +479027.790}
SPL {X  -165.650, Y  +570.048, Z    +0.000, E1   -30.238, E3 +479038.115}
SPL {X  -165.650, Y  +573.110, Z    +0.000, E1   -30.057, E3 +479050.100}
SPL {X  -165.650, Y  +577.587, Z    +0.000, E1   -30.270, E3 +479064.539}
SPL {X  -165.650, Y  +581.190, Z    +0.000, E1   -30.107, E3 +479078.178}
SPL {X  -165.650, Y  +585.053, Z    +0.000, E1   -30.090, E3 +479092.048}
ENDSPLINE

SPLINE
SPL {X  -165.650, Y  +484.445, Z    +0.000, E1   +32.277, E3 +479109.453}
SPL {X  -165.650, Y  +481.524, Z    +0.000, E1   +31.089, E3 +479126.903}
SPL {X  -165.650, Y  +478.014, Z    +0.000, E1   +30.826, E3 +479140.511}
SPL {X  -165.650, Y  +474.473, Z    +0.000, E1   +30.943, E3 +479151.835}
SPL {X  -165.650, Y  +471.826, Z    +0.000, E1   +30.770, E3 +479162.019}
SPL {X  -165.650, Y  +467.753, Z    +0.000, E1   +30.878, E3 +479175.392}
SPL {X  -165.650, Y  +463.837, Z    +0.000, E1   +30.924, E3 +479188.326}
SPL {X  -165.650, Y  +461.106, Z    +0.000, E1   +30.916, E3 +479197.713}
SPL {X  -165.650, Y  +457.156, Z    +0.000, E1   +30.860, E3 +479211.790}
SPL {X  -165.650, Y  +453.156, Z    +0.000, E1   +30.934, E3 +479224.764}
SPL {X  -165.650, Y  +450.433, Z    +0.000, E1   +30.789, E3 +479235.119}
SPL {X  -165.650, Y  +447.097, Z    +0.000, E1   +30.843, E3 +479246.168}
SPL {X  -165.650, Y  +443.673, Z    +0.000, E1   +30.907, E3 +479257.475}
SPL {X  -165.650, Y  +439.486, Z    +0.000, E1   +30.857, E3 +479272.285}
SPL {X  -165.650, Y  +434.043, Z    +0.000, E1   +30.950, E3 +479290.301}
SPL {X  -165.650, Y  +430.419, Z    +0.000, E1   +30.895, E3 +479302.804}
SPL {X  -165.650, Y  +427.340, Z    +0.000, E1   +30.870, E3 +479313.630}
SPL {X  -165.650, Y  +422.641, Z    +0.000, E1   +30.884, E3 +479329.719}
SPL {X  -165.650, Y  +418.489, Z    +0.000, E1   +30.835, E3 +479344.101}
SPL {X  -165.650, Y  +414.127, Z    +0.000, E1   +30.869, E3 +479359.010}
SPL {X  -165.650, Y  +408.547, Z    +0.000, E1   +30.964, E3 +479377.426}
SPL {X  -165.650, Y  +403.421, Z    +0.000, E1   +30.863, E3 +479395.643}
SPL {X  -165.650, Y  +398.147, Z    +0.000, E1   +30.902, E3 +479413.404}
SPL {X  -165.650, Y  +394.694, Z    +0.000, E1   +30.805, E3 +479425.712}
SPL {X  -165.650, Y  +390.331, Z    +0.000, E1   +30.892, E3 +479440.289}
SPL {X  -165.650, Y  +384.849, Z    +0.000, E1   +30.885, E3 +479459.092}
SPL {X  -165.650, Y  +380.752, Z    +0.000, E1   +30.927, E3 +479472.593}
SPL {X  -165.648, Y  +377.739, Z    +0.000, E1   +30.835, E3 +479483.603}
SPL {X  -165.594, Y  +374.183, Z    +0.000, E1   +30.878, E3 +479495.440}
SPL {X  -165.492, Y  +371.263, Z    +0.000, E1   +30.913, E3 +479505.135}
SPL {X  -165.379, Y  +369.027, Z    +0.000, E1   +30.727, E3 +479514.073}
SPL {X  -165.167, Y  +365.866, Z    +0.000, E1   +30.741, E3 +479524.847}
SPL {X  -164.892, Y  +362.671, Z    +0.000, E1   +30.830, E3 +479535.171}
SPL {X  -164.570, Y  +359.612, Z    +0.000, E1   +30.773, E3 +479545.984}
SPL {X  -164.104, Y  +355.923, Z    +0.000, E1   +30.626, E3 +479559.701}
SPL {X  -163.573, Y  +352.353, Z    +0.000, E1   +30.451, E3 +479572.965}
SPL {X  -162.476, Y  +346.230, Z    +0.000, E1   +31.677, E3 +479585.546}
SPL {X  -152.976, Y  +314.952, Z    +0.000, E1   +38.607, E3 +479634.511}
SPL {X  -137.967, Y  +286.821, Z    +0.000, E1   +43.969, E3 +479677.732}
ENDSPLINE

SPLINE
SPL {X  -153.316, Y  +315.777, Z    +0.000, E1   +33.140, E3 +479720.360}
SPL {X  -164.446, Y  +358.564, Z    +0.000, E1   +15.149, E3 +479685.571}
SPL {X  -165.510, Y  +371.680, Z    +0.000, E1    +7.684, E3 +479689.626}
SPL {X  -165.628, Y  +375.818, Z    +0.000, E1    +5.016, E3 +479697.556}
SPL {X  -165.650, Y  +383.362, Z    +0.000, E1    +0.177, E3 +479678.589}
SPL {X  -165.650, Y  +383.923, Z    +0.000, E1    -0.215, E3 +479691.747}
SPL {X  -165.650, Y  +388.083, Z    +0.000, E1    -3.355, E3 +479690.610}
SPL {X  -165.650, Y  +395.510, Z    +0.000, E1    -9.810, E3 +479686.736}
SPL {X  -165.650, Y  +403.066, Z    +0.000, E1   -17.886, E3 +479679.570}
SPL {X  -165.650, Y  +414.811, Z    +0.000, E1   -28.314, E3 +479681.051}
SPL {X  -165.650, Y  +423.479, Z    +0.000, E1   -29.012, E3 +479704.979}
SPL {X  -165.650, Y  +441.276, Z    +0.000, E1   -37.343, E3 +479716.668}
SPL {X  -165.650, Y  +462.890, Z    +0.000, E1   -40.484, E3 +479750.751}
ENDSPLINE

SPLINE
SPL {X  -165.650, Y  +446.920, Z    +0.000, E1   -31.238, E3 +479763.077}
ENDSPLINE

SPLINE
SPL {X  -165.650, Y  +447.935, Z    +0.000, E1   -30.213, E3 +479773.365}
SPL {X  -165.650, Y  +451.020, Z    +0.000, E1   -30.224, E3 +479784.185}
SPL {X  -165.650, Y  +454.519, Z    +0.000, E1   -30.374, E3 +479795.368}
SPL {X  -165.650, Y  +457.429, Z    +0.000, E1   -30.029, E3 +479808.070}
SPL {X  -165.650, Y  +461.678, Z    +0.000, E1   -30.426, E3 +479820.194}
SPL {X  -165.650, Y  +463.853, Z    +0.000, E1   -30.103, E3 +479830.034}
SPL {X  -165.650, Y  +467.246, Z    +0.000, E1   -30.279, E3 +479840.764}
SPL {X  -165.650, Y  +469.780, Z    +0.000, E1   -30.237, E3 +479849.889}
SPL {X  -165.650, Y  +472.566, Z    +0.000, E1   -30.124, E3 +479860.547}
SPL {X  -165.650, Y  +476.540, Z    +0.000, E1   -30.193, E3 +479874.091}
SPL {X  -165.650, Y  +480.320, Z    +0.000, E1   -30.163, E3 +479887.569}
SPL {X  -165.650, Y  +484.477, Z    +0.000, E1   -30.274, E3 +479901.458}
SPL {X  -165.650, Y  +488.041, Z    +0.000, E1   -30.253, E3 +479914.013}
SPL {X  -165.650, Y  +491.281, Z    +0.000, E1   -30.148, E3 +479926.151}
SPL {X  -165.650, Y  +495.051, Z    +0.000, E1   -30.213, E3 +479938.960}
SPL {X  -165.650, Y  +498.418, Z    +0.000, E1   -30.282, E3 +479950.253}
SPL {X  -165.650, Y  +502.421, Z    +0.000, E1   -30.263, E3 +479964.610}
SPL {X  -165.650, Y  +506.344, Z    +0.000, E1   -30.129, E3 +479979.140}
SPL {X  -165.650, Y  +509.866, Z    +0.000, E1   -30.236, E3 +479990.809}
SPL {X  -165.650, Y  +513.685, Z    +0.000, E1   -30.234, E3 +480004.306}
SPL {X  -165.650, Y  +517.104, Z    +0.000, E1   -30.280, E3 +480015.857}
SPL {X  -165.650, Y  +520.621, Z    +0.000, E1   -30.198, E3 +480028.937}
SPL {X  -165.650, Y  +525.344, Z    +0.000, E1   -30.269, E3 +480044.993}
SPL {X  -165.650, Y  +528.152, Z    +0.000, E1   -29.991, E3 +480056.634}
SPL {X  -165.650, Y  +531.783, Z    +0.000, E1   -30.416, E3 +480066.527}
SPL {X  -165.650, Y  +534.115, Z    +0.000, E1   -30.089, E3 +480076.909}
SPL {X  -165.650, Y  +537.522, Z    +0.000, E1   -30.251, E3 +480087.824}
SPL {X  -165.650, Y  +540.621, Z    +0.000, E1   -30.014, E3 +480100.384}
SPL {X  -165.650, Y  +544.944, Z    +0.000, E1   -30.447, E3 +480112.584}
SPL {X  -165.650, Y  +547.199, Z    +0.000, E1   -30.132, E3 +480122.558}
SPL {X  -165.650, Y  +550.512, Z    +0.000, E1   -30.197, E3 +480133.884}
SPL {X  -165.650, Y  +553.852, Z    +0.000, E1   -30.156, E3 +480145.824}
SPL {X  -165.650, Y  +557.277, Z    +0.000, E1   -30.150, E3 +480157.999}
SPL {X  -165.650, Y  +561.168, Z    +0.000, E1   -30.194, E3 +480171.380}
SPL {X  -165.650, Y  +565.528, Z    +0.000, E1   -30.192, E3 +480186.863}
SPL {X  -165.650, Y  +570.048, Z    +0.000, E1   -30.238, E3 +480202.294}
SPL {X  -165.650, Y  +573.110, Z    +0.000, E1   -30.057, E3 +480214.279}
SPL {X  -165.650, Y  +577.587, Z    +0.000, E1   -30.270, E3 +480228.718}
SPL {X  -165.650, Y  +581.190, Z    +0.000, E1   -30.107, E3 +480242.357}
SPL {X  -165.650, Y  +585.053, Z    +0.000, E1   -30.090, E3 +480256.228}
ENDSPLINE

SPLINE
SPL {X  -165.650, Y  +484.445, Z    +0.000, E1   +32.277, E3 +480273.632}
SPL {X  -165.650, Y  +481.524, Z    +0.000, E1   +31.089, E3 +480291.083}
SPL {X  -165.650, Y  +478.014, Z    +0.000, E1   +30.826, E3 +480304.690}
SPL {X  -165.650, Y  +474.473, Z    +0.000, E1   +30.943, E3 +480316.015}
SPL {X  -165.650, Y  +471.826, Z    +0.000, E1   +30.770, E3 +480326.198}
SPL {X  -165.650, Y  +467.753, Z    +0.000, E1   +30.878, E3 +480339.571}
SPL {X  -165.650, Y  +463.837, Z    +0.000, E1   +30.924, E3 +480352.505}
SPL {X  -165.650, Y  +461.106, Z    +0.000, E1   +30.916, E3 +480361.892}
SPL {X  -165.650, Y  +457.156, Z    +0.000, E1   +30.860, E3 +480375.969}
SPL {X  -165.650, Y  +453.156, Z    +0.000, E1   +30.934, E3 +480388.943}
SPL {X  -165.650, Y  +450.433, Z    +0.000, E1   +30.789, E3 +480399.298}
SPL {X  -165.650, Y  +447.097, Z    +0.000, E1   +30.843, E3 +480410.347}
SPL {X  -165.650, Y  +443.673, Z    +0.000, E1   +30.907, E3 +480421.654}
SPL {X  -165.650, Y  +439.486, Z    +0.000, E1   +30.857, E3 +480436.464}
SPL {X  -165.650, Y  +435.146, Z    +0.000, E1   +30.969, E3 +480450.383}
SPL {X  -165.650, Y  +431.607, Z    +0.000, E1   +30.889, E3 +480463.098}
SPL {X  -165.650, Y  +427.340, Z    +0.000, E1   +30.870, E3 +480477.809}
SPL {X  -165.650, Y  +423.901, Z    +0.000, E1   +30.858, E3 +480489.566}
SPL {X  -165.650, Y  +421.437, Z    +0.000, E1   +30.833, E3 +480498.164}
SPL {X  -165.650, Y  +418.489, Z    +0.000, E1   +30.835, E3 +480508.280}
SPL {X  -165.650, Y  +414.127, Z    +0.000, E1   +30.869, E3 +480523.189}
SPL {X  -165.650, Y  +408.547, Z    +0.000, E1   +30.964, E3 +480541.605}
SPL {X  -165.650, Y  +405.433, Z    +0.000, E1   +30.730, E3 +480553.582}
SPL {X  -165.650, Y  +401.473, Z    +0.000, E1   +30.933, E3 +480566.030}
SPL {X  -165.650, Y  +396.018, Z    +0.000, E1   +30.861, E3 +480585.215}
SPL {X  -165.650, Y  +390.331, Z    +0.000, E1   +30.892, E3 +480604.468}
SPL {X  -165.650, Y  +384.849, Z    +0.000, E1   +30.885, E3 +480623.271}
SPL {X  -165.650, Y  +380.752, Z    +0.000, E1   +30.927, E3 +480636.773}
SPL {X  -165.648, Y  +377.739, Z    +0.000, E1   +30.835, E3 +480647.782}
SPL {X  -165.594, Y  +374.183, Z    +0.000, E1   +30.878, E3 +480659.619}
SPL {X  -165.492, Y  +371.263, Z    +0.000, E1   +30.913, E3 +480669.314}
SPL {X  -165.379, Y  +369.027, Z    +0.000, E1   +30.727, E3 +480678.252}
SPL {X  -165.167, Y  +365.866, Z    +0.000, E1   +30.741, E3 +480689.026}
SPL {X  -164.892, Y  +362.671, Z    +0.000, E1   +30.830, E3 +480699.351}
SPL {X  -164.570, Y  +359.612, Z    +0.000, E1   +30.773, E3 +480710.163}
SPL {X  -164.104, Y  +355.923, Z    +0.000, E1   +30.626, E3 +480723.880}
SPL {X  -163.573, Y  +352.353, Z    +0.000, E1   +30.451, E3 +480737.144}
SPL {X  -162.476, Y  +346.230, Z    +0.000, E1   +31.677, E3 +480749.725}
SPL {X  -152.976, Y  +314.952, Z    +0.000, E1   +38.607, E3 +480798.690}
SPL {X  -137.967, Y  +286.821, Z    +0.000, E1   +43.969, E3 +480841.912}
ENDSPLINE

SPLINE
SPL {X  -153.316, Y  +315.777, Z    +0.000, E1   +33.140, E3 +480884.539}
SPL {X  -164.446, Y  +358.564, Z    +0.000, E1   +15.149, E3 +480849.750}
SPL {X  -165.379, Y  +369.025, Z    +0.000, E1    +9.158, E3 +480855.475}
SPL {X  -165.612, Y  +374.969, Z    +0.000, E1    +5.630, E3 +480858.150}
SPL {X  -165.650, Y  +383.362, Z    +0.000, E1    +0.177, E3 +480842.769}
SPL {X  -165.650, Y  +383.923, Z    +0.000, E1    -0.215, E3 +480855.926}
SPL {X  -165.650, Y  +388.083, Z    +0.000, E1    -3.355, E3 +480854.789}
SPL {X  -165.650, Y  +393.983, Z    +0.000, E1    -8.501, E3 +480851.188}
SPL {X  -165.650, Y  +402.241, Z    +0.000, E1   -16.711, E3 +480845.699}
SPL {X  -165.650, Y  +416.345, Z    +0.000, E1   -29.511, E3 +480845.491}
SPL {X  -165.650, Y  +422.331, Z    +0.000, E1   -27.760, E3 +480870.990}
SPL {X  -165.650, Y  +441.276, Z    +0.000, E1   -37.343, E3 +480880.847}
SPL {X  -165.650, Y  +462.890, Z    +0.000, E1   -40.484, E3 +480914.930}
ENDSPLINE

SPLINE
SPL {X  -165.650, Y  +446.920, Z    +0.000, E1   -31.238, E3 +480927.256}
ENDSPLINE

SPLINE
SPL {X  -165.650, Y  +447.935, Z    +0.000, E1   -30.213, E3 +480937.544}
SPL {X  -165.650, Y  +451.020, Z    +0.000, E1   -30.224, E3 +480948.365}
SPL {X  -165.650, Y  +454.519, Z    +0.000, E1   -30.374, E3 +480959.547}
SPL {X  -165.650, Y  +456.542, Z    +0.000, E1   -29.986, E3 +480969.292}
SPL {X  -165.650, Y  +460.618, Z    +0.000, E1   -30.298, E3 +480981.612}
SPL {X  -165.650, Y  +463.853, Z    +0.000, E1   -30.103, E3 +480994.213}
SPL {X  -165.650, Y  +467.246, Z    +0.000, E1   -30.279, E3 +481004.943}
SPL {X  -165.650, Y  +469.780, Z    +0.000, E1   -30.237, E3 +481014.068}
SPL {X  -165.650, Y  +472.566, Z    +0.000, E1   -30.124, E3 +481024.726}
SPL {X  -165.650, Y  +476.540, Z    +0.000, E1   -30.193, E3 +481038.270}
SPL {X  -165.650, Y  +480.320, Z    +0.000, E1   -30.163, E3 +481051.748}
SPL {X  -165.650, Y  +484.477, Z    +0.000, E1   -30.274, E3 +481065.637}
SPL {X  -165.650, Y  +488.041, Z    +0.000, E1   -30.253, E3 +481078.192}
SPL {X  -165.650, Y  +491.281, Z    +0.000, E1   -30.148, E3 +481090.331}
SPL {X  -165.650, Y  +495.051, Z    +0.000, E1   -30.213, E3 +481103.139}
SPL {X  -165.650, Y  +498.418, Z    +0.000, E1   -30.282, E3 +481114.432}
SPL {X  -165.650, Y  +500.833, Z    +0.000, E1   -30.191, E3 +481123.481}
SPL {X  -165.650, Y  +504.246, Z    +0.000, E1   -30.231, E3 +481135.347}
SPL {X  -165.650, Y  +507.017, Z    +0.000, E1   -30.108, E3 +481145.756}
SPL {X  -165.650, Y  +510.660, Z    +0.000, E1   -30.223, E3 +481158.022}
SPL {X  -165.650, Y  +515.918, Z    +0.000, E1   -30.316, E3 +481175.831}
SPL {X  -165.650, Y  +520.621, Z    +0.000, E1   -30.198, E3 +481193.116}
SPL {X  -165.650, Y  +525.344, Z    +0.000, E1   -30.269, E3 +481209.173}
SPL {X  -165.650, Y  +528.152, Z    +0.000, E1   -29.991, E3 +481220.813}
SPL {X  -165.650, Y  +531.783, Z    +0.000, E1   -30.416, E3 +481230.706}
SPL {X  -165.650, Y  +534.115, Z    +0.000, E1   -30.089, E3 +481241.088}
SPL {X  -165.650, Y  +538.363, Z    +0.000, E1   -30.232, E3 +481255.258}
SPL {X  -165.650, Y  +543.650, Z    +0.000, E1   -30.281, E3 +481273.478}
SPL {X  -165.650, Y  +547.199, Z    +0.000, E1   -30.132, E3 +481286.737}
SPL {X  -165.650, Y  +550.512, Z    +0.000, E1   -30.197, E3 +481298.063}
SPL {X  -165.650, Y  +554.908, Z    +0.000, E1   -30.180, E3 +481313.724}
SPL {X  -165.650, Y  +560.243, Z    +0.000, E1   -30.214, E3 +481332.350}
SPL {X  -165.650, Y  +565.528, Z    +0.000, E1   -30.192, E3 +481351.042}
SPL {X  -165.650, Y  +570.048, Z    +0.000, E1   -30.238, E3 +481366.473}
SPL {X  -165.650, Y  +573.110, Z    +0.000, E1   -30.057, E3 +481378.458}
SPL {X  -165.650, Y  +577.587, Z    +0.000, E1   -30.270, E3 +481392.897}
SPL {X  -165.650, Y  +581.190, Z    +0.000, E1   -30.107, E3 +481406.536}
SPL {X  -165.650, Y  +585.053, Z    +0.000, E1   -30.090, E3 +481420.407}
ENDSPLINE

SPLINE
SPL {X  -165.650, Y  +484.445, Z    +0.000, E1   +32.277, E3 +481437.811}
SPL {X  -165.650, Y  +481.524, Z    +0.000, E1   +31.089, E3 +481455.262}
SPL {X  -165.650, Y  +478.014, Z    +0.000, E1   +30.826, E3 +481468.869}
SPL {X  -165.650, Y  +474.473, Z    +0.000, E1   +30.943, E3 +481480.194}
SPL {X  -165.650, Y  +471.826, Z    +0.000, E1   +30.770, E3 +481490.377}
SPL {X  -165.650, Y  +467.753, Z    +0.000, E1   +30.878, E3 +481503.751}
SPL {X  -165.650, Y  +463.837, Z    +0.000, E1   +30.924, E3 +481516.684}
SPL {X  -165.650, Y  +461.106, Z    +0.000, E1   +30.916, E3 +481526.071}
SPL {X  -165.650, Y  +457.156, Z    +0.000, E1   +30.860, E3 +481540.148}
SPL {X  -165.650, Y  +453.156, Z    +0.000, E1   +30.934, E3 +481553.122}
SPL {X  -165.650, Y  +450.433, Z    +0.000, E1   +30.789, E3 +481563.477}
SPL {X  -165.650, Y  +447.097, Z    +0.000, E1   +30.843, E3 +481574.526}
SPL {X  -165.650, Y  +443.673, Z    +0.000, E1   +30.907, E3 +481585.833}
SPL {X  -165.650, Y  +439.486, Z    +0.000, E1   +30.857, E3 +481600.643}
SPL {X  -165.650, Y  +434.043, Z    +0.000, E1   +30.950, E3 +481618.659}
SPL {X  -165.650, Y  +430.419, Z    +0.000, E1   +30.895, E3 +481631.162}
SPL {X  -165.650, Y  +427.340, Z    +0.000, E1   +30.870, E3 +481641.988}
SPL {X  -165.650, Y  +422.641, Z    +0.000, E1   +30.884, E3 +481658.078}
SPL {X  -165.650, Y  +417.366, Z    +0.000, E1   +30.879, E3 +481676.183}
SPL {X  -165.650, Y  +412.139, Z    +0.000, E1   +30.870, E3 +481694.133}
SPL {X  -165.650, Y  +406.834, Z    +0.000, E1   +30.919, E3 +481711.961}
SPL {X  -165.650, Y  +402.516, Z    +0.000, E1   +30.874, E3 +481726.884}
SPL {X  -165.650, Y  +398.147, Z    +0.000, E1   +30.902, E3 +481741.762}
SPL {X  -165.650, Y  +394.694, Z    +0.000, E1   +30.805, E3 +481754.070}
SPL {X  -165.650, Y  +391.522, Z    +0.000, E1   +30.837, E3 +481764.751}
SPL {X  -165.650, Y  +387.533, Z    +0.000, E1   +30.858, E3 +481778.378}
SPL {X  -165.650, Y  +383.627, Z    +0.000, E1   +30.885, E3 +481791.438}
SPL {X  -165.650, Y  +380.752, Z    +0.000, E1   +30.927, E3 +481800.952}
SPL {X  -165.648, Y  +377.739, Z    +0.000, E1   +30.835, E3 +481811.961}
SPL {X  -165.594, Y  +374.183, Z    +0.000, E1   +30.878, E3 +481823.798}
SPL {X  -165.492, Y  +371.263, Z    +0.000, E1   +30.913, E3 +481833.493}
SPL {X  -165.379, Y  +369.027, Z    +0.000, E1   +30.727, E3 +481842.432}
SPL {X  -165.167, Y  +365.866, Z    +0.000, E1   +30.741, E3 +481853.206}
SPL {X  -164.892, Y  +362.671, Z    +0.000, E1   +30.830, E3 +481863.530}
SPL {X  -164.570, Y  +359.612, Z    +0.000, E1   +30.773, E3 +481874.342}
SPL {X  -164.104, Y  +355.923, Z    +0.000, E1   +30.626, E3 +481888.059}
SPL {X  -163.573, Y  +352.353, Z    +0.000, E1   +30.451, E3 +481901.324}
SPL {X  -162.476, Y  +346.230, Z    +0.000, E1   +31.677, E3 +481913.904}
SPL {X  -152.976, Y  +314.952, Z    +0.000, E1   +38.607, E3 +481962.869}
SPL {X  -137.967, Y  +286.821, Z    +0.000, E1   +43.969, E3 +482006.091}
ENDSPLINE

SPLINE
SPL {X  -153.316, Y  +315.777, Z    +0.000, E1   +33.140, E3 +482048.718}
SPL {X  -164.446, Y  +358.564, Z    +0.000, E1   +15.149, E3 +482013.929}
SPL {X  -165.379, Y  +369.025, Z    +0.000, E1    +9.158, E3 +482019.654}
SPL {X  -165.612, Y  +374.969, Z    +0.000, E1    +5.630, E3 +482022.329}
SPL {X  -165.650, Y  +383.362, Z    +0.000, E1    +0.177, E3 +482006.948}
SPL {X  -165.650, Y  +383.923, Z    +0.000, E1    -0.215, E3 +482020.105}
SPL {X  -165.650, Y  +388.083, Z    +0.000, E1    -3.355, E3 +482018.969}
SPL {X  -165.650, Y  +393.983, Z    +0.000, E1    -8.501, E3 +482015.367}
SPL {X  -165.650, Y  +402.241, Z    +0.000, E1   -16.711, E3 +482009.878}
SPL {X  -165.650, Y  +416.345, Z    +0.000, E1   -29.511, E3 +482009.670}
SPL {X  -165.650, Y  +422.331, Z    +0.000, E1   -27.760, E3 +482035.170}
SPL {X  -165.650, Y  +441.276, Z    +0.000, E1   -37.343, E3 +482045.027}
SPL {X  -165.650, Y  +462.890, Z    +0.000, E1   -40.484, E3 +482079.109}
ENDSPLINE

SPLINE
SPL {X  -165.650, Y  +446.920, Z    +0.000, E1   -31.238, E3 +482091.435}
ENDSPLINE

SPLINE
SPL {X  -165.650, Y  +447.935, Z    +0.000, E1   -30.213, E3 +482101.723}
SPL {X  -165.650, Y  +451.020, Z    +0.000, E1   -30.224, E3 +482112.544}
SPL {X  -165.650, Y  +454.519, Z    +0.000, E1   -30.374, E3 +482123.726}
SPL {X  -165.650, Y  +457.429, Z    +0.000, E1   -30.029, E3 +482136.428}
SPL {X  -165.650, Y  +461.678, Z    +0.000, E1   -30.426, E3 +482148.552}
SPL {X  -165.650, Y  +463.853, Z    +0.000, E1   -30.103, E3 +482158.392}
SPL {X  -165.650, Y  +468.397, Z    +0.000, E1   -30.302, E3 +482173.196}
SPL {X  -165.650, Y  +472.566, Z    +0.000, E1   -30.124, E3 +482188.905}
SPL {X  -165.650, Y  +476.540, Z    +0.000, E1   -30.193, E3 +482202.449}
SPL {X  -165.650, Y  +481.042, Z    +0.000, E1   -30.192, E3 +482218.395}
SPL {X  -165.650, Y  +485.236, Z    +0.000, E1   -30.294, E3 +482232.250}
SPL {X  -165.650, Y  +489.057, Z    +0.000, E1   -30.341, E3 +482245.456}
SPL {X  -165.650, Y  +491.647, Z    +0.000, E1   -29.894, E3 +482257.389}
SPL {X  -165.650, Y  +495.051, Z    +0.000, E1   -30.213, E3 +482267.318}
SPL {X  -165.650, Y  +498.418, Z    +0.000, E1   -30.282, E3 +482278.611}
SPL {X  -165.650, Y  +502.421, Z    +0.000, E1   -30.263, E3 +482292.968}
SPL {X  -165.650, Y  +506.344, Z    +0.000, E1   -30.129, E3 +482307.498}
SPL {X  -165.650, Y  +509.866, Z    +0.000, E1   -30.236, E3 +482319.167}
SPL {X  -165.650, Y  +513.685, Z    +0.000, E1   -30.234, E3 +482332.664}
SPL {X  -165.650, Y  +517.919, Z    +0.000, E1   -30.227, E3 +482347.571}
SPL {X  -165.650, Y  +521.521, Z    +0.000, E1   -30.210, E3 +482360.245}
SPL {X  -165.650, Y  +525.344, Z    +0.000, E1   -30.269, E3 +482373.352}
SPL {X  -165.650, Y  +528.152, Z    +0.000, E1   -29.991, E3 +482384.993}
SPL {X  -165.650, Y  +531.783, Z    +0.000, E1   -30.416, E3 +482394.885}
SPL {X  -165.650, Y  +534.115, Z    +0.000, E1   -30.089, E3 +482405.267}
SPL {X  -165.650, Y  +537.522, Z    +0.000, E1   -30.251, E3 +482416.182}
SPL {X  -165.650, Y  +540.621, Z    +0.000, E1   -30.014, E3 +482428.743}
SPL {X  -165.650, Y  +544.944, Z    +0.000, E1   -30.447, E3 +482440.942}
SPL {X  -165.650, Y  +548.549, Z    +0.000, E1   -30.216, E3 +482455.266}
SPL {X  -165.650, Y  +553.092, Z    +0.000, E1   -30.157, E3 +482471.608}
SPL {X  -165.650, Y  +556.274, Z    +0.000, E1   -30.127, E3 +482482.863}
SPL {X  -165.650, Y  +560.243, Z    +0.000, E1   -30.214, E3 +482496.529}
SPL {X  -165.650, Y  +565.528, Z    +0.000, E1   -30.192, E3 +482515.221}
SPL {X  -165.650, Y  +570.048, Z    +0.000, E1   -30.238, E3 +482530.652}
SPL {X  -165.650, Y  +573.110, Z    +0.000, E1   -30.057, E3 +482542.637}
SPL {X  -165.650, Y  +577.587, Z    +0.000, E1   -30.270, E3 +482557.076}
SPL {X  -165.650, Y  +581.190, Z    +0.000, E1   -30.107, E3 +482570.716}
SPL {X  -165.650, Y  +585.053, Z    +0.000, E1   -30.090, E3 +482584.586}
ENDSPLINE

SPLINE
SPL {X  -165.650, Y  +484.445, Z    +0.000, E1   +32.277, E3 +482601.990}
SPL {X  -165.650, Y  +481.524, Z    +0.000, E1   +31.089, E3 +482619.441}
SPL {X  -165.650, Y  +478.014, Z    +0.000, E1   +30.826, E3 +482633.048}
SPL {X  -165.650, Y  +474.473, Z    +0.000, E1   +30.943, E3 +482644.373}
SPL {X  -165.650, Y  +471.826, Z    +0.000, E1   +30.770, E3 +482654.556}
SPL {X  -165.650, Y  +467.753, Z    +0.000, E1   +30.878, E3 +482667.930}
SPL {X  -165.650, Y  +463.837, Z    +0.000, E1   +30.924, E3 +482680.864}
SPL {X  -165.650, Y  +461.106, Z    +0.000, E1   +30.916, E3 +482690.251}
SPL {X  -165.650, Y  +458.435, Z    +0.000, E1   +30.759, E3 +482700.458}
SPL {X  -165.650, Y  +454.220, Z    +0.000, E1   +30.954, E3 +482713.692}
SPL {X  -165.650, Y  +450.433, Z    +0.000, E1   +30.789, E3 +482727.656}
SPL {X  -165.650, Y  +447.097, Z    +0.000, E1   +30.843, E3 +482738.705}
SPL {X  -165.650, Y  +443.673, Z    +0.000, E1   +30.907, E3 +482750.013}
SPL {X  -165.650, Y  +440.976, Z    +0.000, E1   +30.719, E3 +482760.469}
SPL {X  -165.650, Y  +436.324, Z    +0.000, E1   +30.994, E3 +482774.756}
SPL {X  -165.650, Y  +432.765, Z    +0.000, E1   +30.831, E3 +482787.756}
SPL {X  -165.650, Y  +429.309, Z    +0.000, E1   +30.920, E3 +482799.096}
SPL {X  -165.650, Y  +424.918, Z    +0.000, E1   +30.862, E3 +482814.554}
SPL {X  -165.650, Y  +421.437, Z    +0.000, E1   +30.833, E3 +482826.522}
SPL {X  -165.650, Y  +417.366, Z    +0.000, E1   +30.879, E3 +482840.362}
SPL {X  -165.650, Y  +413.181, Z    +0.000, E1   +30.815, E3 +482854.960}
SPL {X  -165.650, Y  +408.547, Z    +0.000, E1   +30.964, E3 +482869.963}
SPL {X  -165.650, Y  +403.421, Z    +0.000, E1   +30.863, E3 +482888.181}
SPL {X  -165.650, Y  +398.147, Z    +0.000, E1   +30.902, E3 +482905.941}
SPL {X  -165.650, Y  +394.694, Z    +0.000, E1   +30.805, E3 +482918.250}
SPL {X  -165.650, Y  +391.522, Z    +0.000, E1   +30.837, E3 +482928.930}
SPL {X  -165.650, Y  +387.533, Z    +0.000, E1   +30.858, E3 +482942.557}
SPL {X  -165.650, Y  +383.627, Z    +0.000, E1   +30.885, E3 +482955.617}
SPL {X  -165.650, Y  +379.886, Z    +0.000, E1   +30.887, E3 +482968.505}
SPL {X  -165.614, Y  +375.058, Z    +0.000, E1   +30.905, E3 +482984.958}
SPL {X  -165.492, Y  +371.263, Z    +0.000, E1   +30.913, E3 +482997.672}
SPL {X  -165.379, Y  +369.027, Z    +0.000, E1   +30.727, E3 +483006.611}
SPL {X  -165.167, Y  +365.866, Z    +0.000, E1   +30.741, E3 +483017.385}
SPL {X  -164.892, Y  +362.671, Z    +0.000, E1   +30.830, E3 +483027.709}
SPL {X  -164.570, Y  +359.612, Z    +0.000, E1   +30.773, E3 +483038.521}
SPL {X  -164.104, Y  +355.923, Z    +0.000, E1   +30.626, E3 +483052.238}
SPL {X  -163.573, Y  +352.353, Z    +0.000, E1   +30.451, E3 +483065.503}
SPL {X  -162.476, Y  +346.230, Z    +0.000, E1   +31.677, E3 +483078.083}
SPL {X  -152.976, Y  +314.952, Z    +0.000, E1   +38.607, E3 +483127.049}
SPL {X  -137.967, Y  +286.821, Z    +0.000, E1   +43.969, E3 +483170.270}
ENDSPLINE

SPLINE
SPL {X  -153.316, Y  +315.777, Z    +0.000, E1   +33.140, E3 +483212.897}
SPL {X  -164.446, Y  +358.564, Z    +0.000, E1   +15.149, E3 +483178.108}
SPL {X  -165.379, Y  +369.025, Z    +0.000, E1    +9.158, E3 +483183.833}
SPL {X  -165.612, Y  +374.969, Z    +0.000, E1    +5.630, E3 +483186.508}
SPL {X  -165.650, Y  +383.362, Z    +0.000, E1    +0.177, E3 +483171.127}
SPL {X  -165.650, Y  +383.923, Z    +0.000, E1    -0.215, E3 +483184.284}
SPL {X  -165.650, Y  +388.083, Z    +0.000, E1    -3.355, E3 +483183.148}
SPL {X  -165.650, Y  +395.510, Z    +0.000, E1    -9.810, E3 +483179.274}
SPL {X  -165.650, Y  +403.066, Z    +0.000, E1   -17.886, E3 +483172.107}
SPL {X  -165.650, Y  +414.811, Z    +0.000, E1   -28.314, E3 +483173.588}
SPL {X  -165.650, Y  +423.479, Z    +0.000, E1   -29.012, E3 +483197.517}
SPL {X  -165.650, Y  +441.276, Z    +0.000, E1   -37.343, E3 +483209.206}
SPL {X  -165.650, Y  +462.890, Z    +0.000, E1   -40.484, E3 +483243.289}
ENDSPLINE

SPLINE
SPL {X  -165.650, Y  +446.920, Z    +0.000, E1   -31.238, E3 +483255.614}
ENDSPLINE

SPLINE
SPL {X  -165.650, Y  +447.935, Z    +0.000, E1   -30.213, E3 +483265.902}
SPL {X  -165.650, Y  +451.020, Z    +0.000, E1   -30.224, E3 +483276.723}
SPL {X  -165.650, Y  +454.519, Z    +0.000, E1   -30.374, E3 +483287.905}
SPL {X  -165.650, Y  +457.429, Z    +0.000, E1   -30.029, E3 +483300.607}
SPL {X  -165.650, Y  +461.678, Z    +0.000, E1   -30.426, E3 +483312.731}
SPL {X  -165.650, Y  +463.853, Z    +0.000, E1   -30.103, E3 +483322.571}
SPL {X  -165.650, Y  +468.397, Z    +0.000, E1   -30.302, E3 +483337.375}
SPL {X  -165.650, Y  +472.566, Z    +0.000, E1   -30.124, E3 +483353.084}
SPL {X  -165.650, Y  +475.265, Z    +0.000, E1   -30.034, E3 +483363.122}
SPL {X  -165.650, Y  +477.862, Z    +0.000, E1   -30.319, E3 +483370.313}
SPL {X  -165.650, Y  +481.042, Z    +0.000, E1   -30.192, E3 +483382.574}
SPL {X  -165.650, Y  +485.236, Z    +0.000, E1   -30.294, E3 +483396.429}
SPL {X  -165.650, Y  +488.041, Z    +0.000, E1   -30.253, E3 +483406.551}
SPL {X  -165.650, Y  +491.281, Z    +0.000, E1   -30.148, E3 +483418.689}
SPL {X  -165.650, Y  +495.051, Z    +0.000, E1   -30.213, E3 +483431.497}
SPL {X  -165.650, Y  +498.418, Z    +0.000, E1   -30.282, E3 +483442.790}
SPL {X  -165.650, Y  +502.421, Z    +0.000, E1   -30.263, E3 +483457.148}
SPL {X  -165.650, Y  +506.344, Z    +0.000, E1   -30.129, E3 +483471.677}
SPL {X  -165.650, Y  +509.866, Z    +0.000, E1   -30.236, E3 +483483.346}
SPL {X  -165.650, Y  +513.685, Z    +0.000, E1   -30.234, E3 +483496.843}
SPL {X  -165.650, Y  +517.104, Z    +0.000, E1   -30.280, E3 +483508.394}
SPL {X  -165.650, Y  +520.621, Z    +0.000, E1   -30.198, E3 +483521.474}
SPL {X  -165.650, Y  +525.344, Z    +0.000, E1   -30.269, E3 +483537.531}
SPL {X  -165.650, Y  +528.152, Z    +0.000, E1   -29.991, E3 +483549.172}
SPL {X  -165.650, Y  +531.783, Z    +0.000, E1   -30.416, E3 +483559.065}
SPL {X  -165.650, Y  +534.115, Z    +0.000, E1   -30.089, E3 +483569.447}
SPL {X  -165.650, Y  +537.522, Z    +0.000, E1   -30.251, E3 +483580.361}
SPL {X  -165.650, Y  +540.621, Z    +0.000, E1   -30.014, E3 +483592.922}
SPL {X  -165.650, Y  +544.944, Z    +0.000, E1   -30.447, E3 +483605.121}
SPL {X  -165.650, Y  +547.199, Z    +0.000, E1   -30.132, E3 +483615.095}
SPL {X  -165.650, Y  +550.512, Z    +0.000, E1   -30.197, E3 +483626.421}
SPL {X  -165.650, Y  +553.852, Z    +0.000, E1   -30.156, E3 +483638.362}
SPL {X  -165.650, Y  +557.277, Z    +0.000, E1   -30.150, E3 +483650.536}
SPL {X  -165.650, Y  +561.168, Z    +0.000, E1   -30.194, E3 +483663.917}
SPL {X  -165.650, Y  +564.449, Z    +0.000, E1   -30.167, E3 +483675.601}
SPL {X  -165.650, Y  +566.935, Z    +0.000, E1   -30.135, E3 +483684.506}
SPL {X  -165.650, Y  +570.048, Z    +0.000, E1   -30.238, E3 +483694.831}
SPL {X  -165.650, Y  +573.110, Z    +0.000, E1   -30.057, E3 +483706.816}
SPL {X  -165.650, Y  +576.497, Z    +0.000, E1   -30.234, E3 +483717.514}
SPL {X  -165.650, Y  +580.354, Z    +0.000, E1   -30.196, E3 +483731.530}
SPL {X  -165.650, Y  +585.053, Z    +0.000, E1   -30.090, E3 +483748.765}
ENDSPLINE

